LIN {X 0,Y 333.799,Z 297.531,A -85,B 0,C 180,E1 6659.656,E2 6659.656} C_VEL
LIN {X 0,Y 333.556,Z 297.579,A -85,B 0,C 180,E1 6657.079,E2 6657.079} C_VEL
LIN {X 0,Y 335.123,Z 301.286,A -85,B 0,C 180,E1 6651.161,E2 6651.161} C_VEL
LIN {X 0,Y 337.536,Z 305.981,A -85,B 0,C 180,E1 6647.598,E2 6647.598} C_VEL
LIN {X 0,Y 340.159,Z 311.065,A -85,B 0,C 180,E1 6644.834,E2 6644.834} C_VEL
LIN {X 0,Y 343.938,Z 318.214,A -85,B 0,C 180,E1 6641.745,E2 6641.745} C_VEL
LIN {X 0,Y 348.405,Z 327.233,A -85,B 0,C 180,E1 6638.757,E2 6638.757} C_VEL
LIN {X 0,Y 349.368,Z 329.534,A -85,B 0,C 180,E1 6638.161,E2 6638.161} C_VEL
LIN {X 0,Y 333.659,Z 514.335,A -85,B 0,C 180,E1 6634.617,E2 6634.617} C_VEL
LIN {X 0,Y 330.211,Z 536.648,A -85,B 0,C 180,E1 6634.047,E2 6634.047} C_VEL
LIN {X 0,Y 325.459,Z 558.771,A -85,B 0,C 180,E1 6633.278,E2 6633.278} C_VEL
LIN {X 0,Y 319.995,Z 578.663,A -85,B 0,C 180,E1 6632.35,E2 6632.35} C_VEL
LIN {X 0,Y 312.977,Z 599.721,A -85,B 0,C 180,E1 6631.082,E2 6631.082} C_VEL
LIN {X 0,Y 305.406,Z 619.136,A -85,B 0,C 180,E1 6629.614,E2 6629.614} C_VEL
LIN {X 0,Y 297.139,Z 637.32,A -85,B 0,C 180,E1 6627.882,E2 6627.882} C_VEL
LIN {X 0,Y 287.577,Z 656.103,A -85,B 0,C 180,E1 6625.662,E2 6625.662} C_VEL
LIN {X 0,Y 278.286,Z 672.56,A -85,B 0,C 180,E1 6623.245,E2 6623.245} C_VEL
LIN {X 0,Y 268.609,Z 688.083,A -85,B 0,C 180,E1 6620.399,E2 6620.399} C_VEL
LIN {X 0,Y 259.107,Z 702.402,A -85,B 0,C 180,E1 6617.152,E2 6617.152} C_VEL
LIN {X 0,Y 249.96,Z 715.337,A -85,B 0,C 180,E1 6613.471,E2 6613.471} C_VEL
LIN {X 0,Y 241.007,Z 727.524,A -85,B 0,C 180,E1 6609.093,E2 6609.093} C_VEL
LIN {X 0,Y 233.429,Z 737.795,A -85,B 0,C 180,E1 6604.429,E2 6604.429} C_VEL
LIN {X 0,Y 227.015,Z 746.575,A -85,B 0,C 180,E1 6599.266,E2 6599.266} C_VEL
LIN {X 0,Y 222.006,Z 753.904,A -85,B 0,C 180,E1 6593.63,E2 6593.63} C_VEL
LIN {X 0,Y 218.703,Z 759.529,A -85,B 0,C 180,E1 6587.836,E2 6587.836} C_VEL
LIN {X 0,Y 216.939,Z 763.245,A -85,B 0,C 180,E1 6582.24,E2 6582.24} C_VEL
LIN {X 0,Y 216.215,Z 765.602,A -85,B 0,C 180,E1 6576.639,E2 6576.639} C_VEL
LIN {X 0,Y 216.046,Z 766.465,A -85,B 0,C 180,E1 6571.856,E2 6571.856} C_VEL
LIN {X 0,Y 216.061,Z 766.392,A -85,B 0,C 180,E1 6567.082,E2 6567.082} C_VEL
LIN {X 0,Y 216.332,Z 765.111,A -85,B 0,C 180,E1 6561.763,E2 6561.763} C_VEL
LIN {X 0,Y 217.229,Z 762.561,A -85,B 0,C 180,E1 6556.424,E2 6556.424} C_VEL
LIN {X 0,Y 219.54,Z 757.995,A -85,B 0,C 180,E1 6550.305,E2 6550.305} C_VEL
LIN {X 0,Y 223.351,Z 751.966,A -85,B 0,C 180,E1 6544.549,E2 6544.549} C_VEL
LIN {X 0,Y 228.596,Z 744.406,A -85,B 0,C 180,E1 6539.221,E2 6539.221} C_VEL
LIN {X 0,Y 235.447,Z 735.08,A -85,B 0,C 180,E1 6534.125,E2 6534.125} C_VEL
LIN {X 0,Y 243.448,Z 724.408,A -85,B 0,C 180,E1 6529.541,E2 6529.541} C_VEL
LIN {X 0,Y 252.267,Z 712.209,A -85,B 0,C 180,E1 6525.451,E2 6525.451} C_VEL
LIN {X 0,Y 262.23,Z 697.898,A -85,B 0,C 180,E1 6521.642,E2 6521.642} C_VEL
LIN {X 0,Y 272.029,Z 682.985,A -85,B 0,C 180,E1 6518.476,E2 6518.476} C_VEL
LIN {X 0,Y 281.596,Z 667.003,A -85,B 0,C 180,E1 6515.776,E2 6515.776} C_VEL
LIN {X 0,Y 291.404,Z 649.061,A -85,B 0,C 180,E1 6513.335,E2 6513.335} C_VEL
LIN {X 0,Y 300.317,Z 630.949,A -85,B 0,C 180,E1 6511.356,E2 6511.356} C_VEL
LIN {X 0,Y 308.467,Z 611.849,A -85,B 0,C 180,E1 6509.696,E2 6509.696} C_VEL
LIN {X 0,Y 316.13,Z 591.143,A -85,B 0,C 180,E1 6508.259,E2 6508.259} C_VEL
LIN {X 0,Y 322.47,Z 570.714,A -85,B 0,C 180,E1 6507.145,E2 6507.145} C_VEL
LIN {X 0,Y 327.778,Z 549.297,A -85,B 0,C 180,E1 6506.26,E2 6506.26} C_VEL
LIN {X 0,Y 332.035,Z 527,A -85,B 0,C 180,E1 6505.584,E2 6505.584} C_VEL
LIN {X 0,Y 334.766,Z 504.932,A -85,B 0,C 180,E1 6505.085,E2 6505.085} C_VEL
LIN {X 0,Y 335.935,Z 491.115,A -85,B 0,C 180,E1 6504.815,E2 6504.815} C_VEL
LIN {X 0,Y 336.181,Z 483.557,A -85,B 0,C 180,E1 6504.514,E2 6504.514} C_VEL
LIN {X 0,Y 335.511,Z 463.894,A -85,B 0,C 180,E1 6503.143,E2 6503.143} C_VEL
LIN {X 0,Y 335.792,Z 457.395,A -85,B 0,C 180,E1 6502.899,E2 6502.899} C_VEL
LIN {X 0,Y 346.51,Z 334.247,A -85,B 0,C 180,E1 6500.568,E2 6500.568} C_VEL
LIN {X 0,Y 342.284,Z 325.412,A -85,B 0,C 180,E1 6497.598,E2 6497.598} C_VEL
LIN {X 0,Y 338.735,Z 318.442,A -85,B 0,C 180,E1 6494.531,E2 6494.531} C_VEL
LIN {X 0,Y 335.95,Z 312.735,A -85,B 0,C 180,E1 6491.329,E2 6491.329} C_VEL
LIN {X 0,Y 333.881,Z 308.598,A -85,B 0,C 180,E1 6487.745,E2 6487.745} C_VEL
LIN {X 0,Y 332.812,Z 305.703,A -85,B 0,C 180,E1 6482.239,E2 6482.239} C_VEL
LIN {X 0,Y 333.175,Z 306.116,A -85,B 0,C 180,E1 6479.656,E2 6479.656} C_VEL
LIN {X 0,Y 335.748,Z 309.602,A -85,B 0,C 180,E1 6474.275,E2 6474.275} C_VEL
LIN {X 0,Y 338.837,Z 314.734,A -85,B 0,C 180,E1 6470.66,E2 6470.66} C_VEL
LIN {X 0,Y 342.068,Z 320.176,A -85,B 0,C 180,E1 6467.851,E2 6467.851} C_VEL
LIN {X 0,Y 346.16,Z 327.49,A -85,B 0,C 180,E1 6464.933,E2 6464.933} C_VEL
LIN {X 0,Y 348.005,Z 331.065,A -85,B 0,C 180,E1 6463.762,E2 6463.762} C_VEL
LIN {X 0,Y 331.369,Z 511.396,A -85,B 0,C 180,E1 6460.174,E2 6460.174} C_VEL
LIN {X 0,Y 327.681,Z 534.66,A -85,B 0,C 180,E1 6459.571,E2 6459.571} C_VEL
LIN {X 0,Y 322.798,Z 557.073,A -85,B 0,C 180,E1 6458.798,E2 6458.798} C_VEL
LIN {X 0,Y 316.826,Z 578.359,A -85,B 0,C 180,E1 6457.813,E2 6457.813} C_VEL
LIN {X 0,Y 309.169,Z 600.967,A -85,B 0,C 180,E1 6456.465,E2 6456.465} C_VEL
LIN {X 0,Y 301.055,Z 621.475,A -85,B 0,C 180,E1 6454.919,E2 6454.919} C_VEL
LIN {X 0,Y 292.123,Z 640.891,A -85,B 0,C 180,E1 6453.074,E2 6453.074} C_VEL
LIN {X 0,Y 281.948,Z 660.722,A -85,B 0,C 180,E1 6450.733,E2 6450.733} C_VEL
LIN {X 0,Y 272.269,Z 677.831,A -85,B 0,C 180,E1 6448.225,E2 6448.225} C_VEL
LIN {X 0,Y 262.16,Z 694.192,A -85,B 0,C 180,E1 6445.249,E2 6445.249} C_VEL
LIN {X 0,Y 251.99,Z 709.754,A -85,B 0,C 180,E1 6441.759,E2 6441.759} C_VEL
LIN {X 0,Y 242.523,Z 723.441,A -85,B 0,C 180,E1 6437.908,E2 6437.908} C_VEL
LIN {X 0,Y 232.836,Z 737.179,A -85,B 0,C 180,E1 6433.06,E2 6433.06} C_VEL
LIN {X 0,Y 225.094,Z 748.311,A -85,B 0,C 180,E1 6428.128,E2 6428.128} C_VEL
LIN {X 0,Y 218.579,Z 757.937,A -85,B 0,C 180,E1 6422.667,E2 6422.667} C_VEL
LIN {X 0,Y 213.445,Z 766.429,A -85,B 0,C 180,E1 6416.529,E2 6416.529} C_VEL
LIN {X 0,Y 210.416,Z 772.403,A -85,B 0,C 180,E1 6410.878,E2 6410.878} C_VEL
LIN {X 0,Y 208.638,Z 777.202,A -85,B 0,C 180,E1 6404.713,E2 6404.713} C_VEL
LIN {X 0,Y 208.082,Z 779.88,A -85,B 0,C 180,E1 6399.682,E2 6399.682} C_VEL
LIN {X 0,Y 207.995,Z 781.502,A -85,B 0,C 180,E1 6394.687,E2 6394.687} C_VEL
LIN {X 0,Y 208.03,Z 782.018,A -85,B 0,C 180,E1 6389.725,E2 6389.725} C_VEL
LIN {X 0,Y 207.994,Z 781.35,A -85,B 0,C 180,E1 6384.76,E2 6384.76} C_VEL
LIN {X 0,Y 208.096,Z 779.747,A -85,B 0,C 180,E1 6380.04,E2 6380.04} C_VEL
LIN {X 0,Y 208.804,Z 776.674,A -85,B 0,C 180,E1 6374.446,E2 6374.446} C_VEL
LIN {X 0,Y 210.701,Z 771.73,A -85,B 0,C 180,E1 6368.449,E2 6368.449} C_VEL
LIN {X 0,Y 214.139,Z 765.22,A -85,B 0,C 180,E1 6362.468,E2 6362.468} C_VEL
LIN {X 0,Y 219.122,Z 757.046,A -85,B 0,C 180,E1 6356.801,E2 6356.801} C_VEL
LIN {X 0,Y 226.148,Z 746.654,A -85,B 0,C 180,E1 6351.112,E2 6351.112} C_VEL
LIN {X 0,Y 234.128,Z 735.335,A -85,B 0,C 180,E1 6346.226,E2 6346.226} C_VEL
LIN {X 0,Y 243.307,Z 722.206,A -85,B 0,C 180,E1 6341.738,E2 6341.738} C_VEL
LIN {X 0,Y 253.129,Z 707.933,A -85,B 0,C 180,E1 6337.817,E2 6337.817} C_VEL
LIN {X 0,Y 263.1,Z 692.584,A -85,B 0,C 180,E1 6334.448,E2 6334.448} C_VEL
LIN {X 0,Y 273.875,Z 674.84,A -85,B 0,C 180,E1 6331.322,E2 6331.322} C_VEL
LIN {X 0,Y 284.002,Z 656.771,A -85,B 0,C 180,E1 6328.765,E2 6328.765} C_VEL
LIN {X 0,Y 293.417,Z 637.944,A -85,B 0,C 180,E1 6326.636,E2 6326.636} C_VEL
LIN {X 0,Y 302.733,Z 617.038,A -85,B 0,C 180,E1 6324.737,E2 6324.737} C_VEL
LIN {X 0,Y 310.741,Z 596.454,A -85,B 0,C 180,E1 6323.244,E2 6323.244} C_VEL
LIN {X 0,Y 317.653,Z 575.154,A -85,B 0,C 180,E1 6322.035,E2 6322.035} C_VEL
LIN {X 0,Y 323.863,Z 551.917,A -85,B 0,C 180,E1 6321.013,E2 6321.013} C_VEL
LIN {X 0,Y 328.488,Z 529.683,A -85,B 0,C 180,E1 6320.29,E2 6320.29} C_VEL
LIN {X 0,Y 331.75,Z 506.604,A -85,B 0,C 180,E1 6319.732,E2 6319.732} C_VEL
LIN {X 0,Y 347.863,Z 330.818,A -85,B 0,C 180,E1 6316.238,E2 6316.238} C_VEL
LIN {X 0,Y 343.256,Z 322.384,A -85,B 0,C 180,E1 6313.175,E2 6313.175} C_VEL
LIN {X 0,Y 339.741,Z 316.374,A -85,B 0,C 180,E1 6310.342,E2 6310.342} C_VEL
LIN {X 0,Y 337.54,Z 312.774,A -85,B 0,C 180,E1 6308.174,E2 6308.174} C_VEL
LIN {X 0,Y 335.255,Z 309.045,A -85,B 0,C 180,E1 6305.305,E2 6305.305} C_VEL
LIN {X 0,Y 332.793,Z 305.429,A -85,B 0,C 180,E1 6299.483,E2 6299.483} C_VEL
LIN {X 0,Y 332.58,Z 305.538,A -85,B 0,C 180,E1 6297.07,E2 6297.07} C_VEL
LIN {X 0,Y 334.018,Z 309.105,A -85,B 0,C 180,E1 6291.392,E2 6291.392} C_VEL
LIN {X 0,Y 336.286,Z 313.689,A -85,B 0,C 180,E1 6287.9,E2 6287.9} C_VEL
LIN {X 0,Y 338.827,Z 318.787,A -85,B 0,C 180,E1 6285.124,E2 6285.124} C_VEL
LIN {X 0,Y 342.557,Z 326.138,A -85,B 0,C 180,E1 6281.977,E2 6281.977} C_VEL
LIN {X 0,Y 346.368,Z 334.145,A -85,B 0,C 180,E1 6279.331,E2 6279.331} C_VEL
LIN {X 0,Y 330.595,Z 514.238,A -85,B 0,C 180,E1 6275.897,E2 6275.897} C_VEL
LIN {X 0,Y 327.044,Z 536.692,A -85,B 0,C 180,E1 6275.332,E2 6275.332} C_VEL
LIN {X 0,Y 322.156,Z 558.903,A -85,B 0,C 180,E1 6274.573,E2 6274.573} C_VEL
LIN {X 0,Y 316.376,Z 579.413,A -85,B 0,C 180,E1 6273.629,E2 6273.629} C_VEL
LIN {X 0,Y 309.189,Z 600.314,A -85,B 0,C 180,E1 6272.38,E2 6272.38} C_VEL
LIN {X 0,Y 301.428,Z 619.632,A -85,B 0,C 180,E1 6270.93,E2 6270.93} C_VEL
LIN {X 0,Y 292.82,Z 638.021,A -85,B 0,C 180,E1 6269.19,E2 6269.19} C_VEL
LIN {X 0,Y 282.759,Z 657.106,A -85,B 0,C 180,E1 6266.932,E2 6266.932} C_VEL
LIN {X 0,Y 272.873,Z 674.008,A -85,B 0,C 180,E1 6264.432,E2 6264.432} C_VEL
LIN {X 0,Y 262.899,Z 689.345,A -85,B 0,C 180,E1 6261.576,E2 6261.576} C_VEL
LIN {X 0,Y 252.519,Z 704.237,A -85,B 0,C 180,E1 6258.105,E2 6258.105} C_VEL
LIN {X 0,Y 242.805,Z 717.433,A -85,B 0,C 180,E1 6254.231,E2 6254.231} C_VEL
LIN {X 0,Y 233.844,Z 728.953,A -85,B 0,C 180,E1 6249.892,E2 6249.892} C_VEL
LIN {X 0,Y 225.636,Z 739.428,A -85,B 0,C 180,E1 6244.863,E2 6244.863} C_VEL
LIN {X 0,Y 219.071,Z 748.046,A -85,B 0,C 180,E1 6239.532,E2 6239.532} C_VEL
LIN {X 0,Y 213.953,Z 755.074,A -85,B 0,C 180,E1 6233.696,E2 6233.696} C_VEL
LIN {X 0,Y 210.496,Z 760.607,A -85,B 0,C 180,E1 6227.412,E2 6227.412} C_VEL
LIN {X 0,Y 208.819,Z 764.143,A -85,B 0,C 180,E1 6221.601,E2 6221.601} C_VEL
LIN {X 0,Y 208.183,Z 766.083,A -85,B 0,C 180,E1 6216.065,E2 6216.065} C_VEL
LIN {X 0,Y 208.05,Z 766.82,A -85,B 0,C 180,E1 6211.101,E2 6211.101} C_VEL
LIN {X 0,Y 208.1,Z 766.558,A -85,B 0,C 180,E1 6205.867,E2 6205.867} C_VEL
LIN {X 0,Y 208.5,Z 764.977,A -85,B 0,C 180,E1 6200.338,E2 6200.338} C_VEL
LIN {X 0,Y 209.774,Z 762.063,A -85,B 0,C 180,E1 6194.52,E2 6194.52} C_VEL
LIN {X 0,Y 212.497,Z 757.324,A -85,B 0,C 180,E1 6188.469,E2 6188.469} C_VEL
LIN {X 0,Y 216.927,Z 750.912,A -85,B 0,C 180,E1 6182.554,E2 6182.554} C_VEL
LIN {X 0,Y 223.082,Z 742.845,A -85,B 0,C 180,E1 6176.945,E2 6176.945} C_VEL
LIN {X 0,Y 230.422,Z 733.396,A -85,B 0,C 180,E1 6171.964,E2 6171.964} C_VEL
LIN {X 0,Y 239.579,Z 721.646,A -85,B 0,C 180,E1 6167.137,E2 6167.137} C_VEL
LIN {X 0,Y 249.147,Z 709.054,A -85,B 0,C 180,E1 6163.083,E2 6163.083} C_VEL
LIN {X 0,Y 258.622,Z 695.757,A -85,B 0,C 180,E1 6159.706,E2 6159.706} C_VEL
LIN {X 0,Y 269.416,Z 679.56,A -85,B 0,C 180,E1 6156.427,E2 6156.427} C_VEL
LIN {X 0,Y 279.594,Z 662.962,A -85,B 0,C 180,E1 6153.755,E2 6153.755} C_VEL
LIN {X 0,Y 289.138,Z 645.535,A -85,B 0,C 180,E1 6151.527,E2 6151.527} C_VEL
LIN {X 0,Y 298.371,Z 626.661,A -85,B 0,C 180,E1 6149.591,E2 6149.591} C_VEL
LIN {X 0,Y 306.714,Z 607.269,A -85,B 0,C 180,E1 6147.997,E2 6147.997} C_VEL
LIN {X 0,Y 313.949,Z 587.306,A -85,B 0,C 180,E1 6146.708,E2 6146.708} C_VEL
LIN {X 0,Y 320.465,Z 565.899,A -85,B 0,C 180,E1 6145.623,E2 6145.623} C_VEL
LIN {X 0,Y 325.353,Z 545.873,A -85,B 0,C 180,E1 6144.851,E2 6144.851} C_VEL
LIN {X 0,Y 329.463,Z 523.359,A -85,B 0,C 180,E1 6144.215,E2 6144.215} C_VEL
LIN {X 0,Y 332.202,Z 499.849,A -85,B 0,C 180,E1 6143.708,E2 6143.708} C_VEL
LIN {X 0,Y 335.792,Z 457.395,A -85,B 0,C 180,E1 6142.899,E2 6142.899} C_VEL
LIN {X 0,Y 336.087,Z 449.841,A -85,B 0,C 180,E1 6142.594,E2 6142.594} C_VEL
LIN {X 0,Y 335.695,Z 430.195,A -85,B 0,C 180,E1 6141.211,E2 6141.211} C_VEL
LIN {X 0,Y 336.035,Z 423.697,A -85,B 0,C 180,E1 6140.971,E2 6140.971} C_VEL
LIN {X 0,Y 343.619,Z 339.193,A -85,B 0,C 180,E1 6139.373,E2 6139.373} C_VEL
LIN {X 0,Y 339.767,Z 330.925,A -85,B 0,C 180,E1 6136.41,E2 6136.41} C_VEL
LIN {X 0,Y 336.405,Z 323.949,A -85,B 0,C 180,E1 6133.143,E2 6133.143} C_VEL
LIN {X 0,Y 334.367,Z 319.872,A -85,B 0,C 180,E1 6130.51,E2 6130.51} C_VEL
LIN {X 0,Y 332.808,Z 316.439,A -85,B 0,C 180,E1 6127.522,E2 6127.522} C_VEL
LIN {X 0,Y 331.836,Z 313.655,A -85,B 0,C 180,E1 6122.245,E2 6122.245} C_VEL
LIN {X 0,Y 332.158,Z 313.997,A -85,B 0,C 180,E1 6119.828,E2 6119.828} C_VEL
LIN {X 0,Y 334.577,Z 317.402,A -85,B 0,C 180,E1 6114.513,E2 6114.513} C_VEL
LIN {X 0,Y 337.577,Z 322.568,A -85,B 0,C 180,E1 6110.883,E2 6110.883} C_VEL
LIN {X 0,Y 340.629,Z 327.878,A -85,B 0,C 180,E1 6108.143,E2 6108.143} C_VEL
LIN {X 0,Y 344.745,Z 335.474,A -85,B 0,C 180,E1 6105.127,E2 6105.127} C_VEL
LIN {X 0,Y 345.018,Z 336.358,A -85,B 0,C 180,E1 6104.922,E2 6104.922} C_VEL
LIN {X 0,Y 328.43,Z 511.584,A -85,B 0,C 180,E1 6101.468,E2 6101.468} C_VEL
LIN {X 0,Y 324.675,Z 534.746,A -85,B 0,C 180,E1 6100.878,E2 6100.878} C_VEL
LIN {X 0,Y 319.704,Z 557.076,A -85,B 0,C 180,E1 6100.124,E2 6100.124} C_VEL
LIN {X 0,Y 313.499,Z 578.698,A -85,B 0,C 180,E1 6099.14,E2 6099.14} C_VEL
LIN {X 0,Y 305.987,Z 600.374,A -85,B 0,C 180,E1 6097.873,E2 6097.873} C_VEL
LIN {X 0,Y 297.498,Z 621.33,A -85,B 0,C 180,E1 6096.322,E2 6096.322} C_VEL
LIN {X 0,Y 288.555,Z 640.271,A -85,B 0,C 180,E1 6094.554,E2 6094.554} C_VEL
LIN {X 0,Y 278.341,Z 659.691,A -85,B 0,C 180,E1 6092.307,E2 6092.307} C_VEL
LIN {X 0,Y 268.308,Z 676.872,A -85,B 0,C 180,E1 6089.829,E2 6089.829} C_VEL
LIN {X 0,Y 257.656,Z 693.579,A -85,B 0,C 180,E1 6086.828,E2 6086.828} C_VEL
LIN {X 0,Y 247.511,Z 708.558,A -85,B 0,C 180,E1 6083.501,E2 6083.501} C_VEL
LIN {X 0,Y 236.977,Z 723.105,A -85,B 0,C 180,E1 6079.415,E2 6079.415} C_VEL
LIN {X 0,Y 226.773,Z 736.859,A -85,B 0,C 180,E1 6074.509,E2 6074.509} C_VEL
LIN {X 0,Y 218.548,Z 747.992,A -85,B 0,C 180,E1 6069.487,E2 6069.487} C_VEL
LIN {X 0,Y 211.578,Z 757.626,A -85,B 0,C 180,E1 6063.891,E2 6063.891} C_VEL
LIN {X 0,Y 206.155,Z 765.916,A -85,B 0,C 180,E1 6057.748,E2 6057.748} C_VEL
LIN {X 0,Y 202.844,Z 771.832,A -85,B 0,C 180,E1 6052,E2 6052} C_VEL
LIN {X 0,Y 200.741,Z 776.906,A -85,B 0,C 180,E1 6045.306,E2 6045.306} C_VEL
LIN {X 0,Y 200.102,Z 779.586,A -85,B 0,C 180,E1 6040.072,E2 6040.072} C_VEL
LIN {X 0,Y 199.997,Z 781.211,A -85,B 0,C 180,E1 6034.875,E2 6034.875} C_VEL
LIN {X 0,Y 200.035,Z 781.727,A -85,B 0,C 180,E1 6029.714,E2 6029.714} C_VEL
LIN {X 0,Y 199.997,Z 781.058,A -85,B 0,C 180,E1 6024.55,E2 6024.55} C_VEL
LIN {X 0,Y 200.12,Z 779.451,A -85,B 0,C 180,E1 6019.638,E2 6019.638} C_VEL
LIN {X 0,Y 200.923,Z 776.376,A -85,B 0,C 180,E1 6013.819,E2 6013.819} C_VEL
LIN {X 0,Y 202.97,Z 771.536,A -85,B 0,C 180,E1 6007.71,E2 6007.71} C_VEL
LIN {X 0,Y 206.57,Z 765.244,A -85,B 0,C 180,E1 6001.684,E2 6001.684} C_VEL
LIN {X 0,Y 211.866,Z 757.155,A -85,B 0,C 180,E1 5995.835,E2 5995.835} C_VEL
LIN {X 0,Y 218.913,Z 747.401,A -85,B 0,C 180,E1 5990.252,E2 5990.252} C_VEL
LIN {X 0,Y 227.219,Z 736.196,A -85,B 0,C 180,E1 5985.247,E2 5985.247} C_VEL
LIN {X 0,Y 237.229,Z 722.653,A -85,B 0,C 180,E1 5980.471,E2 5980.471} C_VEL
LIN {X 0,Y 247.5,Z 708.444,A -85,B 0,C 180,E1 5976.495,E2 5976.495} C_VEL
LIN {X 0,Y 257.831,Z 693.165,A -85,B 0,C 180,E1 5973.111,E2 5973.111} C_VEL
LIN {X 0,Y 269.302,Z 675.009,A -85,B 0,C 180,E1 5969.899,E2 5969.899} C_VEL
LIN {X 0,Y 279.396,Z 657.645,A -85,B 0,C 180,E1 5967.442,E2 5967.442} C_VEL
LIN {X 0,Y 289.323,Z 638.454,A -85,B 0,C 180,E1 5965.277,E2 5965.277} C_VEL
LIN {X 0,Y 298.891,Z 617.672,A -85,B 0,C 180,E1 5963.402,E2 5963.402} C_VEL
LIN {X 0,Y 307.154,Z 597.004,A -85,B 0,C 180,E1 5961.918,E2 5961.918} C_VEL
LIN {X 0,Y 314.28,Z 575.687,A -85,B 0,C 180,E1 5960.721,E2 5960.721} C_VEL
LIN {X 0,Y 320.498,Z 553.187,A -85,B 0,C 180,E1 5959.738,E2 5959.738} C_VEL
LIN {X 0,Y 325.186,Z 531.346,A -85,B 0,C 180,E1 5959.032,E2 5959.032} C_VEL
LIN {X 0,Y 328.718,Z 507.683,A -85,B 0,C 180,E1 5958.459,E2 5958.459} C_VEL
LIN {X 0,Y 344.865,Z 335.93,A -85,B 0,C 180,E1 5955.064,E2 5955.064} C_VEL
LIN {X 0,Y 340.775,Z 328.253,A -85,B 0,C 180,E1 5952.11,E2 5952.11} C_VEL
LIN {X 0,Y 337.662,Z 322.863,A -85,B 0,C 180,E1 5949.373,E2 5949.373} C_VEL
LIN {X 0,Y 335.93,Z 320.014,A -85,B 0,C 180,E1 5947.525,E2 5947.525} C_VEL
LIN {X 0,Y 334.034,Z 316.781,A -85,B 0,C 180,E1 5944.98,E2 5944.98} C_VEL
LIN {X 0,Y 331.789,Z 313.328,A -85,B 0,C 180,E1 5939.309,E2 5939.309} C_VEL
LIN {X 0,Y 331.602,Z 313.552,A -85,B 0,C 180,E1 5936.955,E2 5936.955} C_VEL
LIN {X 0,Y 332.92,Z 316.923,A -85,B 0,C 180,E1 5931.624,E2 5931.624} C_VEL
LIN {X 0,Y 335.067,Z 321.465,A -85,B 0,C 180,E1 5928.165,E2 5928.165} C_VEL
LIN {X 0,Y 337.851,Z 327.149,A -85,B 0,C 180,E1 5925.08,E2 5925.08} C_VEL
LIN {X 0,Y 341.177,Z 334.101,A -85,B 0,C 180,E1 5922.21,E2 5922.21} C_VEL
LIN {X 0,Y 343.483,Z 339.338,A -85,B 0,C 180,E1 5920.5,E2 5920.5} C_VEL
LIN {X 0,Y 327.692,Z 514.168,A -85,B 0,C 180,E1 5917.199,E2 5917.199} C_VEL
LIN {X 0,Y 324.064,Z 536.634,A -85,B 0,C 180,E1 5916.645,E2 5916.645} C_VEL
LIN {X 0,Y 319.02,Z 559.031,A -85,B 0,C 180,E1 5915.895,E2 5915.895} C_VEL
LIN {X 0,Y 313.304,Z 578.886,A -85,B 0,C 180,E1 5915.001,E2 5915.001} C_VEL
LIN {X 0,Y 305.946,Z 599.91,A -85,B 0,C 180,E1 5913.775,E2 5913.775} C_VEL
LIN {X 0,Y 297.989,Z 619.319,A -85,B 0,C 180,E1 5912.349,E2 5912.349} C_VEL
LIN {X 0,Y 289.115,Z 637.808,A -85,B 0,C 180,E1 5910.631,E2 5910.631} C_VEL
LIN {X 0,Y 278.971,Z 656.588,A -85,B 0,C 180,E1 5908.447,E2 5908.447} C_VEL
LIN {X 0,Y 268.903,Z 673.331,A -85,B 0,C 180,E1 5906.012,E2 5906.012} C_VEL
LIN {X 0,Y 258.528,Z 688.828,A -85,B 0,C 180,E1 5903.168,E2 5903.168} C_VEL
LIN {X 0,Y 247.721,Z 703.818,A -85,B 0,C 180,E1 5899.714,E2 5899.714} C_VEL
LIN {X 0,Y 237.84,Z 716.674,A -85,B 0,C 180,E1 5895.96,E2 5895.96} C_VEL
LIN {X 0,Y 228.528,Z 728.154,A -85,B 0,C 180,E1 5891.683,E2 5891.683} C_VEL
LIN {X 0,Y 220.104,Z 738.408,A -85,B 0,C 180,E1 5886.842,E2 5886.842} C_VEL
LIN {X 0,Y 212.871,Z 747.186,A -85,B 0,C 180,E1 5881.423,E2 5881.423} C_VEL
LIN {X 0,Y 207.136,Z 754.504,A -85,B 0,C 180,E1 5875.442,E2 5875.442} C_VEL
LIN {X 0,Y 203.268,Z 760.122,A -85,B 0,C 180,E1 5869.242,E2 5869.242} C_VEL
LIN {X 0,Y 201.156,Z 763.836,A -85,B 0,C 180,E1 5863.217,E2 5863.217} C_VEL
LIN {X 0,Y 200.244,Z 766.248,A -85,B 0,C 180,E1 5856.882,E2 5856.882} C_VEL
LIN {X 0,Y 200.057,Z 767.072,A -85,B 0,C 180,E1 5851.66,E2 5851.66} C_VEL
LIN {X 0,Y 200.084,Z 766.953,A -85,B 0,C 180,E1 5846.562,E2 5846.562} C_VEL
LIN {X 0,Y 200.446,Z 765.589,A -85,B 0,C 180,E1 5840.815,E2 5840.815} C_VEL
LIN {X 0,Y 201.594,Z 762.998,A -85,B 0,C 180,E1 5835.054,E2 5835.054} C_VEL
LIN {X 0,Y 204.259,Z 758.589,A -85,B 0,C 180,E1 5828.763,E2 5828.763} C_VEL
LIN {X 0,Y 208.692,Z 752.568,A -85,B 0,C 180,E1 5822.617,E2 5822.617} C_VEL
LIN {X 0,Y 214.701,Z 744.975,A -85,B 0,C 180,E1 5816.957,E2 5816.957} C_VEL
LIN {X 0,Y 222.774,Z 735.198,A -85,B 0,C 180,E1 5811.403,E2 5811.403} C_VEL
LIN {X 0,Y 231.704,Z 724.431,A -85,B 0,C 180,E1 5806.678,E2 5806.678} C_VEL
LIN {X 0,Y 241.435,Z 712.168,A -85,B 0,C 180,E1 5802.512,E2 5802.512} C_VEL
LIN {X 0,Y 251.697,Z 698.574,A -85,B 0,C 180,E1 5798.869,E2 5798.869} C_VEL
LIN {X 0,Y 262.271,Z 683.632,A -85,B 0,C 180,E1 5795.682,E2 5795.682} C_VEL
LIN {X 0,Y 272.782,Z 667.21,A -85,B 0,C 180,E1 5792.928,E2 5792.928} C_VEL
LIN {X 0,Y 283.216,Z 649.242,A -85,B 0,C 180,E1 5790.527,E2 5790.527} C_VEL
LIN {X 0,Y 292.828,Z 630.745,A -85,B 0,C 180,E1 5788.557,E2 5788.557} C_VEL
LIN {X 0,Y 301.231,Z 612.009,A -85,B 0,C 180,E1 5786.977,E2 5786.977} C_VEL
LIN {X 0,Y 309.278,Z 591.313,A -85,B 0,C 180,E1 5785.585,E2 5785.585} C_VEL
LIN {X 0,Y 315.519,Z 572.179,A -85,B 0,C 180,E1 5784.569,E2 5784.569} C_VEL
LIN {X 0,Y 321.306,Z 550.248,A -85,B 0,C 180,E1 5783.68,E2 5783.68} C_VEL
LIN {X 0,Y 325.784,Z 528.283,A -85,B 0,C 180,E1 5783.028,E2 5783.028} C_VEL
LIN {X 0,Y 328.747,Z 505.867,A -85,B 0,C 180,E1 5782.529,E2 5782.529} C_VEL
LIN {X 0,Y 336.035,Z 423.697,A -85,B 0,C 180,E1 5780.971,E2 5780.971} C_VEL
LIN {X 0,Y 336.398,Z 416.144,A -85,B 0,C 180,E1 5780.671,E2 5780.671} C_VEL
LIN {X 0,Y 336.265,Z 396.516,A -85,B 0,C 180,E1 5779.282,E2 5779.282} C_VEL
LIN {X 0,Y 336.643,Z 390.022,A -85,B 0,C 180,E1 5779.038,E2 5779.038} C_VEL
LIN {X 0,Y 340.866,Z 344.206,A -85,B 0,C 180,E1 5778.16,E2 5778.16} C_VEL
LIN {X 0,Y 337.728,Z 337.382,A -85,B 0,C 180,E1 5775.541,E2 5775.541} C_VEL
LIN {X 0,Y 334.984,Z 331.384,A -85,B 0,C 180,E1 5772.673,E2 5772.673} C_VEL
LIN {X 0,Y 333.17,Z 327.584,A -85,B 0,C 180,E1 5770.199,E2 5770.199} C_VEL
LIN {X 0,Y 331.723,Z 324.266,A -85,B 0,C 180,E1 5767.273,E2 5767.273} C_VEL
LIN {X 0,Y 330.873,Z 321.562,A -85,B 0,C 180,E1 5762.078,E2 5762.078} C_VEL
LIN {X 0,Y 331.25,Z 322.126,A -85,B 0,C 180,E1 5759.481,E2 5759.481} C_VEL
LIN {X 0,Y 333.465,Z 325.323,A -85,B 0,C 180,E1 5754.667,E2 5754.667} C_VEL
LIN {X 0,Y 336.242,Z 330.251,A -85,B 0,C 180,E1 5751.191,E2 5751.191} C_VEL
LIN {X 0,Y 339.197,Z 335.579,A -85,B 0,C 180,E1 5748.437,E2 5748.437} C_VEL
LIN {X 0,Y 342.193,Z 341.477,A -85,B 0,C 180,E1 5746.105,E2 5746.105} C_VEL
LIN {X 0,Y 325.674,Z 511.674,A -85,B 0,C 180,E1 5742.787,E2 5742.787} C_VEL
LIN {X 0,Y 321.84,Z 534.834,A -85,B 0,C 180,E1 5742.208,E2 5742.208} C_VEL
LIN {X 0,Y 316.721,Z 557.318,A -85,B 0,C 180,E1 5741.464,E2 5741.464} C_VEL
LIN {X 0,Y 310.684,Z 577.955,A -85,B 0,C 180,E1 5740.548,E2 5740.548} C_VEL
LIN {X 0,Y 302.596,Z 600.8,A -85,B 0,C 180,E1 5739.241,E2 5739.241} C_VEL
LIN {X 0,Y 294.291,Z 620.797,A -85,B 0,C 180,E1 5737.789,E2 5737.789} C_VEL
LIN {X 0,Y 285.025,Z 639.97,A -85,B 0,C 180,E1 5736.036,E2 5736.036} C_VEL
LIN {X 0,Y 274.753,Z 659.006,A -85,B 0,C 180,E1 5733.875,E2 5733.875} C_VEL
LIN {X 0,Y 264.222,Z 676.482,A -85,B 0,C 180,E1 5731.39,E2 5731.39} C_VEL
LIN {X 0,Y 253.047,Z 693.41,A -85,B 0,C 180,E1 5728.373,E2 5728.373} C_VEL
LIN {X 0,Y 242.016,Z 709.037,A -85,B 0,C 180,E1 5724.884,E2 5724.884} C_VEL
LIN {X 0,Y 231.31,Z 723.162,A -85,B 0,C 180,E1 5720.869,E2 5720.869} C_VEL
LIN {X 0,Y 220.86,Z 736.537,A -85,B 0,C 180,E1 5716.037,E2 5716.037} C_VEL
LIN {X 0,Y 212.13,Z 747.673,A -85,B 0,C 180,E1 5710.931,E2 5710.931} C_VEL
LIN {X 0,Y 204.677,Z 757.314,A -85,B 0,C 180,E1 5705.199,E2 5705.199} C_VEL
LIN {X 0,Y 198.818,Z 765.612,A -85,B 0,C 180,E1 5698.867,E2 5698.867} C_VEL
LIN {X 0,Y 195.1,Z 771.707,A -85,B 0,C 180,E1 5692.711,E2 5692.711} C_VEL
LIN {X 0,Y 192.859,Z 776.608,A -85,B 0,C 180,E1 5685.948,E2 5685.948} C_VEL
LIN {X 0,Y 192.122,Z 779.333,A -85,B 0,C 180,E1 5680.391,E2 5680.391} C_VEL
LIN {X 0,Y 192.001,Z 780.919,A -85,B 0,C 180,E1 5675.079,E2 5675.079} C_VEL
LIN {X 0,Y 192.04,Z 781.437,A -85,B 0,C 180,E1 5669.702,E2 5669.702} C_VEL
LIN {X 0,Y 192.003,Z 780.765,A -85,B 0,C 180,E1 5664.322,E2 5664.322} C_VEL
LIN {X 0,Y 192.15,Z 779.156,A -85,B 0,C 180,E1 5659.203,E2 5659.203} C_VEL
LIN {X 0,Y 193.061,Z 776.077,A -85,B 0,C 180,E1 5653.141,E2 5653.141} C_VEL
LIN {X 0,Y 195.335,Z 771.232,A -85,B 0,C 180,E1 5646.788,E2 5646.788} C_VEL
LIN {X 0,Y 199.502,Z 764.6,A -85,B 0,C 180,E1 5640.254,E2 5640.254} C_VEL
LIN {X 0,Y 205.304,Z 756.419,A -85,B 0,C 180,E1 5634.239,E2 5634.239} C_VEL
LIN {X 0,Y 213.329,Z 746.011,A -85,B 0,C 180,E1 5628.277,E2 5628.277} C_VEL
LIN {X 0,Y 222.29,Z 734.686,A -85,B 0,C 180,E1 5623.226,E2 5623.226} C_VEL
LIN {X 0,Y 232.148,Z 721.954,A -85,B 0,C 180,E1 5618.781,E2 5618.781} C_VEL
LIN {X 0,Y 242.611,Z 708.087,A -85,B 0,C 180,E1 5614.905,E2 5614.905} C_VEL
LIN {X 0,Y 253.361,Z 692.8,A -85,B 0,C 180,E1 5611.527,E2 5611.527} C_VEL
LIN {X 0,Y 265.149,Z 674.785,A -85,B 0,C 180,E1 5608.368,E2 5608.368} C_VEL
LIN {X 0,Y 275.678,Z 657.227,A -85,B 0,C 180,E1 5605.914,E2 5605.914} C_VEL
LIN {X 0,Y 285.772,Z 638.233,A -85,B 0,C 180,E1 5603.807,E2 5603.807} C_VEL
LIN {X 0,Y 295.842,Z 616.85,A -85,B 0,C 180,E1 5601.921,E2 5601.921} C_VEL
LIN {X 0,Y 304.195,Z 596.402,A -85,B 0,C 180,E1 5600.489,E2 5600.489} C_VEL
LIN {X 0,Y 311.486,Z 574.931,A -85,B 0,C 180,E1 5599.317,E2 5599.317} C_VEL
LIN {X 0,Y 317.988,Z 551.533,A -85,B 0,C 180,E1 5598.333,E2 5598.333} C_VEL
LIN {X 0,Y 322.851,Z 528.982,A -85,B 0,C 180,E1 5597.636,E2 5597.636} C_VEL
LIN {X 0,Y 326.173,Z 505.964,A -85,B 0,C 180,E1 5597.103,E2 5597.103} C_VEL
LIN {X 0,Y 342.026,Z 341.243,A -85,B 0,C 180,E1 5593.89,E2 5593.89} C_VEL
LIN {X 0,Y 338.444,Z 334.385,A -85,B 0,C 180,E1 5591.071,E2 5591.071} C_VEL
LIN {X 0,Y 335.302,Z 328.678,A -85,B 0,C 180,E1 5587.97,E2 5587.97} C_VEL
LIN {X 0,Y 332.934,Z 324.653,A -85,B 0,C 180,E1 5584.823,E2 5584.823} C_VEL
LIN {X 0,Y 330.813,Z 321.277,A -85,B 0,C 180,E1 5579.307,E2 5579.307} C_VEL
LIN {X 0,Y 330.626,Z 321.472,A -85,B 0,C 180,E1 5577.053,E2 5577.053} C_VEL
LIN {X 0,Y 331.862,Z 324.857,A -85,B 0,C 180,E1 5571.772,E2 5571.772} C_VEL
LIN {X 0,Y 333.8,Z 329.103,A -85,B 0,C 180,E1 5568.51,E2 5568.51} C_VEL
LIN {X 0,Y 336.521,Z 334.865,A -85,B 0,C 180,E1 5565.371,E2 5565.371} C_VEL
LIN {X 0,Y 339.644,Z 341.745,A -85,B 0,C 180,E1 5562.57,E2 5562.57} C_VEL
LIN {X 0,Y 340.732,Z 344.478,A -85,B 0,C 180,E1 5561.696,E2 5561.696} C_VEL
LIN {X 0,Y 324.968,Z 514.053,A -85,B 0,C 180,E1 5558.525,E2 5558.525} C_VEL
LIN {X 0,Y 321.257,Z 536.567,A -85,B 0,C 180,E1 5557.981,E2 5557.981} C_VEL
LIN {X 0,Y 316.26,Z 558.423,A -85,B 0,C 180,E1 5557.271,E2 5557.271} C_VEL
LIN {X 0,Y 310.416,Z 578.356,A -85,B 0,C 180,E1 5556.399,E2 5556.399} C_VEL
LIN {X 0,Y 302.89,Z 599.504,A -85,B 0,C 180,E1 5555.198,E2 5555.198} C_VEL
LIN {X 0,Y 294.776,Z 618.901,A -85,B 0,C 180,E1 5553.807,E2 5553.807} C_VEL
LIN {X 0,Y 285.785,Z 637.229,A -85,B 0,C 180,E1 5552.144,E2 5552.144} C_VEL
LIN {X 0,Y 275.357,Z 656.115,A -85,B 0,C 180,E1 5549.997,E2 5549.997} C_VEL
LIN {X 0,Y 265.142,Z 672.624,A -85,B 0,C 180,E1 5547.638,E2 5547.638} C_VEL
LIN {X 0,Y 254.416,Z 688.236,A -85,B 0,C 180,E1 5544.827,E2 5544.827} C_VEL
LIN {X 0,Y 243.74,Z 702.644,A -85,B 0,C 180,E1 5541.581,E2 5541.581} C_VEL
LIN {X 0,Y 233.321,Z 715.635,A -85,B 0,C 180,E1 5537.846,E2 5537.846} C_VEL
LIN {X 0,Y 222.962,Z 727.912,A -85,B 0,C 180,E1 5533.322,E2 5533.322} C_VEL
LIN {X 0,Y 214.01,Z 738.27,A -85,B 0,C 180,E1 5528.416,E2 5528.416} C_VEL
LIN {X 0,Y 206.246,Z 747.101,A -85,B 0,C 180,E1 5522.885,E2 5522.885} C_VEL
LIN {X 0,Y 200.019,Z 754.515,A -85,B 0,C 180,E1 5516.736,E2 5516.736} C_VEL
LIN {X 0,Y 195.749,Z 760.222,A -85,B 0,C 180,E1 5510.324,E2 5510.324} C_VEL
LIN {X 0,Y 193.358,Z 763.979,A -85,B 0,C 180,E1 5504.065,E2 5504.065} C_VEL
LIN {X 0,Y 192.322,Z 766.415,A -85,B 0,C 180,E1 5497.768,E2 5497.768} C_VEL
LIN {X 0,Y 192.066,Z 767.338,A -85,B 0,C 180,E1 5492.088,E2 5492.088} C_VEL
LIN {X 0,Y 192.078,Z 767.285,A -85,B 0,C 180,E1 5487.016,E2 5487.016} C_VEL
LIN {X 0,Y 192.425,Z 766.096,A -85,B 0,C 180,E1 5481.032,E2 5481.032} C_VEL
LIN {X 0,Y 193.609,Z 763.555,A -85,B 0,C 180,E1 5474.958,E2 5474.958} C_VEL
LIN {X 0,Y 196.506,Z 759.129,A -85,B 0,C 180,E1 5468.196,E2 5468.196} C_VEL
LIN {X 0,Y 201.198,Z 753.188,A -85,B 0,C 180,E1 5461.83,E2 5461.83} C_VEL
LIN {X 0,Y 207.61,Z 745.578,A -85,B 0,C 180,E1 5455.931,E2 5455.931} C_VEL
LIN {X 0,Y 216.323,Z 735.627,A -85,B 0,C 180,E1 5450.109,E2 5450.109} C_VEL
LIN {X 0,Y 225.816,Z 724.748,A -85,B 0,C 180,E1 5445.252,E2 5445.252} C_VEL
LIN {X 0,Y 236,Z 712.479,A -85,B 0,C 180,E1 5441.048,E2 5441.048} C_VEL
LIN {X 0,Y 247.283,Z 698.084,A -85,B 0,C 180,E1 5437.201,E2 5437.201} C_VEL
LIN {X 0,Y 258.232,Z 683.079,A -85,B 0,C 180,E1 5434.048,E2 5434.048} C_VEL
LIN {X 0,Y 268.965,Z 666.813,A -85,B 0,C 180,E1 5431.362,E2 5431.362} C_VEL
LIN {X 0,Y 279.574,Z 649.001,A -85,B 0,C 180,E1 5429.026,E2 5429.026} C_VEL
LIN {X 0,Y 289.264,Z 630.82,A -85,B 0,C 180,E1 5427.122,E2 5427.122} C_VEL
LIN {X 0,Y 298.072,Z 611.64,A -85,B 0,C 180,E1 5425.536,E2 5425.536} C_VEL
LIN {X 0,Y 306.311,Z 590.834,A -85,B 0,C 180,E1 5424.173,E2 5424.173} C_VEL
LIN {X 0,Y 313.032,Z 570.585,A -85,B 0,C 180,E1 5423.134,E2 5423.134} C_VEL
LIN {X 0,Y 318.632,Z 549.413,A -85,B 0,C 180,E1 5422.31,E2 5422.31} C_VEL
LIN {X 0,Y 323.172,Z 527.21,A -85,B 0,C 180,E1 5421.674,E2 5421.674} C_VEL
LIN {X 0,Y 326.128,Z 505.091,A -85,B 0,C 180,E1 5421.192,E2 5421.192} C_VEL
LIN {X 0,Y 336.643,Z 390.022,A -85,B 0,C 180,E1 5419.038,E2 5419.038} C_VEL
LIN {X 0,Y 337.059,Z 382.472,A -85,B 0,C 180,E1 5418.735,E2 5418.735} C_VEL
LIN {X 0,Y 337.224,Z 362.849,A -85,B 0,C 180,E1 5417.348,E2 5417.348} C_VEL
LIN {X 0,Y 337.665,Z 356.354,A -85,B 0,C 180,E1 5417.112,E2 5417.112} C_VEL
LIN {X 0,Y 338.297,Z 349.512,A -85,B 0,C 180,E1 5416.97,E2 5416.97} C_VEL
LIN {X 0,Y 335.771,Z 343.804,A -85,B 0,C 180,E1 5414.662,E2 5414.662} C_VEL
LIN {X 0,Y 333.25,Z 338.137,A -85,B 0,C 180,E1 5411.773,E2 5411.773} C_VEL
LIN {X 0,Y 331.984,Z 335.295,A -85,B 0,C 180,E1 5409.885,E2 5409.885} C_VEL
LIN {X 0,Y 330.68,Z 332.15,A -85,B 0,C 180,E1 5407.122,E2 5407.122} C_VEL
LIN {X 0,Y 329.897,Z 329.512,A -85,B 0,C 180,E1 5402.085,E2 5402.085} C_VEL
LIN {X 0,Y 330.225,Z 330.007,A -85,B 0,C 180,E1 5399.653,E2 5399.653} C_VEL
LIN {X 0,Y 332.355,Z 333.243,A -85,B 0,C 180,E1 5394.822,E2 5394.822} C_VEL
LIN {X 0,Y 334.918,Z 337.934,A -85,B 0,C 180,E1 5391.502,E2 5391.502} C_VEL
LIN {X 0,Y 337.976,Z 343.622,A -85,B 0,C 180,E1 5388.568,E2 5388.568} C_VEL
LIN {X 0,Y 339.482,Z 346.907,A -85,B 0,C 180,E1 5387.301,E2 5387.301} C_VEL
LIN {X 0,Y 323.094,Z 511.762,A -85,B 0,C 180,E1 5384.127,E2 5384.127} C_VEL
LIN {X 0,Y 319.182,Z 534.928,A -85,B 0,C 180,E1 5383.561,E2 5383.561} C_VEL
LIN {X 0,Y 313.937,Z 557.483,A -85,B 0,C 180,E1 5382.832,E2 5382.832} C_VEL
LIN {X 0,Y 307.645,Z 578.511,A -85,B 0,C 180,E1 5381.917,E2 5381.917} C_VEL
LIN {X 0,Y 299.791,Z 600.212,A -85,B 0,C 180,E1 5380.705,E2 5380.705} C_VEL
LIN {X 0,Y 290.884,Z 621.167,A -85,B 0,C 180,E1 5379.215,E2 5379.215} C_VEL
LIN {X 0,Y 281.385,Z 640.258,A -85,B 0,C 180,E1 5377.495,E2 5377.495} C_VEL
LIN {X 0,Y 270.631,Z 659.547,A -85,B 0,C 180,E1 5375.325,E2 5375.325} C_VEL
LIN {X 0,Y 260.342,Z 676.093,A -85,B 0,C 180,E1 5372.997,E2 5372.997} C_VEL
LIN {X 0,Y 248.6,Z 693.287,A -85,B 0,C 180,E1 5369.964,E2 5369.964} C_VEL
LIN {X 0,Y 237.297,Z 708.698,A -85,B 0,C 180,E1 5366.538,E2 5366.538} C_VEL
LIN {X 0,Y 226.419,Z 722.44,A -85,B 0,C 180,E1 5362.641,E2 5362.641} C_VEL
LIN {X 0,Y 215.107,Z 736.217,A -85,B 0,C 180,E1 5357.65,E2 5357.65} C_VEL
LIN {X 0,Y 205.715,Z 747.532,A -85,B 0,C 180,E1 5352.373,E2 5352.373} C_VEL
LIN {X 0,Y 197.554,Z 757.427,A -85,B 0,C 180,E1 5346.309,E2 5346.309} C_VEL
LIN {X 0,Y 191.084,Z 765.944,A -85,B 0,C 180,E1 5339.462,E2 5339.462} C_VEL
LIN {X 0,Y 187.142,Z 772.031,A -85,B 0,C 180,E1 5332.955,E2 5332.955} C_VEL
LIN {X 0,Y 184.855,Z 776.652,A -85,B 0,C 180,E1 5326.012,E2 5326.012} C_VEL
LIN {X 0,Y 184.118,Z 779.24,A -85,B 0,C 180,E1 5320.323,E2 5320.323} C_VEL
LIN {X 0,Y 184.007,Z 780.826,A -85,B 0,C 180,E1 5314.363,E2 5314.363} C_VEL
LIN {X 0,Y 184.043,Z 781.099,A -85,B 0,C 180,E1 5309.066,E2 5309.066} C_VEL
LIN {X 0,Y 184.014,Z 780.4,A -85,B 0,C 180,E1 5303.761,E2 5303.761} C_VEL
LIN {X 0,Y 184.216,Z 778.738,A -85,B 0,C 180,E1 5298.415,E2 5298.415} C_VEL
LIN {X 0,Y 185.392,Z 775.387,A -85,B 0,C 180,E1 5291.772,E2 5291.772} C_VEL
LIN {X 0,Y 188.083,Z 770.391,A -85,B 0,C 180,E1 5285.168,E2 5285.168} C_VEL
LIN {X 0,Y 192.806,Z 763.55,A -85,B 0,C 180,E1 5278.416,E2 5278.416} C_VEL
LIN {X 0,Y 198.905,Z 755.684,A -85,B 0,C 180,E1 5272.539,E2 5272.539} C_VEL
LIN {X 0,Y 207.574,Z 745.157,A -85,B 0,C 180,E1 5266.465,E2 5266.465} C_VEL
LIN {X 0,Y 217.135,Z 733.769,A -85,B 0,C 180,E1 5261.361,E2 5261.361} C_VEL
LIN {X 0,Y 227.567,Z 720.897,A -85,B 0,C 180,E1 5256.906,E2 5256.906} C_VEL
LIN {X 0,Y 239.18,Z 705.997,A -85,B 0,C 180,E1 5252.836,E2 5252.836} C_VEL
LIN {X 0,Y 250.122,Z 691.015,A -85,B 0,C 180,E1 5249.608,E2 5249.608} C_VEL
LIN {X 0,Y 261.412,Z 674.217,A -85,B 0,C 180,E1 5246.738,E2 5246.738} C_VEL
LIN {X 0,Y 272.163,Z 656.8,A -85,B 0,C 180,E1 5244.347,E2 5244.347} C_VEL
LIN {X 0,Y 282.545,Z 637.765,A -85,B 0,C 180,E1 5242.277,E2 5242.277} C_VEL
LIN {X 0,Y 292.473,Z 617.216,A -85,B 0,C 180,E1 5240.499,E2 5240.499} C_VEL
LIN {X 0,Y 301.015,Z 596.818,A -85,B 0,C 180,E1 5239.096,E2 5239.096} C_VEL
LIN {X 0,Y 308.465,Z 575.468,A -85,B 0,C 180,E1 5237.95,E2 5237.95} C_VEL
LIN {X 0,Y 314.991,Z 552.696,A -85,B 0,C 180,E1 5237.005,E2 5237.005} C_VEL
LIN {X 0,Y 319.889,Z 530.631,A -85,B 0,C 180,E1 5236.33,E2 5236.33} C_VEL
LIN {X 0,Y 323.449,Z 507.345,A -85,B 0,C 180,E1 5235.791,E2 5235.791} C_VEL
LIN {X 0,Y 339.327,Z 346.52,A -85,B 0,C 180,E1 5232.689,E2 5232.689} C_VEL
LIN {X 0,Y 335.796,Z 339.699,A -85,B 0,C 180,E1 5229.598,E2 5229.598} C_VEL
LIN {X 0,Y 333.631,Z 335.82,A -85,B 0,C 180,E1 5227.231,E2 5227.231} C_VEL
LIN {X 0,Y 331.731,Z 332.389,A -85,B 0,C 180,E1 5224.494,E2 5224.494} C_VEL
LIN {X 0,Y 329.813,Z 329.176,A -85,B 0,C 180,E1 5219.131,E2 5219.131} C_VEL
LIN {X 0,Y 329.646,Z 329.533,A -85,B 0,C 180,E1 5216.87,E2 5216.87} C_VEL
LIN {X 0,Y 330.773,Z 332.673,A -85,B 0,C 180,E1 5212.007,E2 5212.007} C_VEL
LIN {X 0,Y 332.63,Z 336.956,A -85,B 0,C 180,E1 5208.733,E2 5208.733} C_VEL
LIN {X 0,Y 335.148,Z 342.543,A -85,B 0,C 180,E1 5205.707,E2 5205.707} C_VEL
LIN {X 0,Y 337.981,Z 349.024,A -85,B 0,C 180,E1 5203.058,E2 5203.058} C_VEL
LIN {X 0,Y 338.118,Z 349.793,A -85,B 0,C 180,E1 5202.907,E2 5202.907} C_VEL
LIN {X 0,Y 322.394,Z 514.167,A -85,B 0,C 180,E1 5199.869,E2 5199.869} C_VEL
LIN {X 0,Y 318.601,Z 536.633,A -85,B 0,C 180,E1 5199.336,E2 5199.336} C_VEL
LIN {X 0,Y 313.48,Z 558.547,A -85,B 0,C 180,E1 5198.641,E2 5198.641} C_VEL
LIN {X 0,Y 307.314,Z 579.1,A -85,B 0,C 180,E1 5197.76,E2 5197.76} C_VEL
LIN {X 0,Y 299.624,Z 600.092,A -85,B 0,C 180,E1 5196.586,E2 5196.586} C_VEL
LIN {X 0,Y 290.891,Z 620.3,A -85,B 0,C 180,E1 5195.149,E2 5195.149} C_VEL
LIN {X 0,Y 281.571,Z 638.717,A -85,B 0,C 180,E1 5193.486,E2 5193.486} C_VEL
LIN {X 0,Y 271.039,Z 657.113,A -85,B 0,C 180,E1 5191.396,E2 5191.396} C_VEL
LIN {X 0,Y 260.192,Z 674.092,A -85,B 0,C 180,E1 5188.972,E2 5188.972} C_VEL
LIN {X 0,Y 249.153,Z 689.497,A -85,B 0,C 180,E1 5186.168,E2 5186.168} C_VEL
LIN {X 0,Y 237.269,Z 704.764,A -85,B 0,C 180,E1 5182.64,E2 5182.64} C_VEL
LIN {X 0,Y 226.216,Z 718.008,A -85,B 0,C 180,E1 5178.709,E2 5178.709} C_VEL
LIN {X 0,Y 216.069,Z 729.34,A -85,B 0,C 180,E1 5174.325,E2 5174.325} C_VEL
LIN {X 0,Y 206.361,Z 739.905,A -85,B 0,C 180,E1 5169.039,E2 5169.039} C_VEL
LIN {X 0,Y 198.39,Z 748.577,A -85,B 0,C 180,E1 5163.321,E2 5163.321} C_VEL
LIN {X 0,Y 192.192,Z 755.455,A -85,B 0,C 180,E1 5157.175,E2 5157.175} C_VEL
LIN {X 0,Y 187.649,Z 761.106,A -85,B 0,C 180,E1 5150.263,E2 5150.263} C_VEL
LIN {X 0,Y 185.269,Z 764.728,A -85,B 0,C 180,E1 5143.736,E2 5143.736} C_VEL
LIN {X 0,Y 184.277,Z 766.895,A -85,B 0,C 180,E1 5137.169,E2 5137.169} C_VEL
LIN {X 0,Y 184.067,Z 767.653,A -85,B 0,C 180,E1 5131.813,E2 5131.813} C_VEL
LIN {X 0,Y 184.103,Z 767.534,A -85,B 0,C 180,E1 5126.263,E2 5126.263} C_VEL
LIN {X 0,Y 184.555,Z 766.175,A -85,B 0,C 180,E1 5120.017,E2 5120.017} C_VEL
LIN {X 0,Y 185.964,Z 763.586,A -85,B 0,C 180,E1 5113.765,E2 5113.765} C_VEL
LIN {X 0,Y 189.217,Z 759.083,A -85,B 0,C 180,E1 5106.846,E2 5106.846} C_VEL
LIN {X 0,Y 194.299,Z 753.17,A -85,B 0,C 180,E1 5100.396,E2 5100.396} C_VEL
LIN {X 0,Y 201.493,Z 745.221,A -85,B 0,C 180,E1 5094.16,E2 5094.16} C_VEL
LIN {X 0,Y 210.211,Z 735.811,A -85,B 0,C 180,E1 5088.614,E2 5088.614} C_VEL
LIN {X 0,Y 220.077,Z 725.064,A -85,B 0,C 180,E1 5083.751,E2 5083.751} C_VEL
LIN {X 0,Y 230.712,Z 712.806,A -85,B 0,C 180,E1 5079.521,E2 5079.521} C_VEL
LIN {X 0,Y 242.443,Z 698.419,A -85,B 0,C 180,E1 5075.666,E2 5075.666} C_VEL
LIN {X 0,Y 253.775,Z 683.439,A -85,B 0,C 180,E1 5072.529,E2 5072.529} C_VEL
LIN {X 0,Y 264.616,Z 667.531,A -85,B 0,C 180,E1 5069.919,E2 5069.919} C_VEL
LIN {X 0,Y 275.753,Z 649.417,A -85,B 0,C 180,E1 5067.562,E2 5067.562} C_VEL
LIN {X 0,Y 285.691,Z 631.276,A -85,B 0,C 180,E1 5065.688,E2 5065.688} C_VEL
LIN {X 0,Y 294.707,Z 612.161,A -85,B 0,C 180,E1 5064.131,E2 5064.131} C_VEL
LIN {X 0,Y 303.13,Z 591.477,A -85,B 0,C 180,E1 5062.796,E2 5062.796} C_VEL
LIN {X 0,Y 309.648,Z 572.36,A -85,B 0,C 180,E1 5061.826,E2 5061.826} C_VEL
LIN {X 0,Y 315.686,Z 550.472,A -85,B 0,C 180,E1 5060.978,E2 5060.978} C_VEL
LIN {X 0,Y 320.384,Z 528.412,A -85,B 0,C 180,E1 5060.351,E2 5060.351} C_VEL
LIN {X 0,Y 323.493,Z 506.016,A -85,B 0,C 180,E1 5059.868,E2 5059.868} C_VEL
LIN {X 0,Y 337.665,Z 356.354,A -85,B 0,C 180,E1 5057.112,E2 5057.112} C_VEL
LIN {X 0,Y 337.664,Z 354.032,A -85,B 0,C 180,E1 5056.923,E2 5056.923} C_VEL
LIN {X 0,Y 337.212,Z 352.045,A -85,B 0,C 180,E1 5056.458,E2 5056.458} C_VEL
LIN {X 0,Y 336.2,Z 350.71,A -85,B 0,C 180,E1 5055.632,E2 5055.632} C_VEL
LIN {X 0,Y 333.714,Z 349.633,A -85,B 0,C 180,E1 5053.557,E2 5053.557} C_VEL
LIN {X 0,Y 333.443,Z 349.174,A -85,B 0,C 180,E1 5053.268,E2 5053.268} C_VEL
LIN {X 0,Y 331.218,Z 343.78,A -85,B 0,C 180,E1 5050.238,E2 5050.238} C_VEL
LIN {X 0,Y 329.573,Z 339.928,A -85,B 0,C 180,E1 5046.795,E2 5046.795} C_VEL
LIN {X 0,Y 328.935,Z 337.424,A -85,B 0,C 180,E1 5041.916,E2 5041.916} C_VEL
LIN {X 0,Y 329.32,Z 338.144,A -85,B 0,C 180,E1 5039.304,E2 5039.304} C_VEL
LIN {X 0,Y 331.198,Z 341.041,A -85,B 0,C 180,E1 5035.064,E2 5035.064} C_VEL
LIN {X 0,Y 333.597,Z 345.615,A -85,B 0,C 180,E1 5031.815,E2 5031.815} C_VEL
LIN {X 0,Y 336.459,Z 351.167,A -85,B 0,C 180,E1 5028.95,E2 5028.95} C_VEL
LIN {X 0,Y 336.911,Z 352.508,A -85,B 0,C 180,E1 5028.513,E2 5028.513} C_VEL
LIN {X 0,Y 320.681,Z 511.967,A -85,B 0,C 180,E1 5025.486,E2 5025.486} C_VEL
LIN {X 0,Y 316.706,Z 535.018,A -85,B 0,C 180,E1 5024.936,E2 5024.936} C_VEL
LIN {X 0,Y 311.631,Z 556.631,A -85,B 0,C 180,E1 5024.263,E2 5024.263} C_VEL
LIN {X 0,Y 305.21,Z 577.771,A -85,B 0,C 180,E1 5023.374,E2 5023.374} C_VEL
LIN {X 0,Y 296.768,Z 600.64,A -85,B 0,C 180,E1 5022.131,E2 5022.131} C_VEL
LIN {X 0,Y 288.071,Z 620.638,A -85,B 0,C 180,E1 5020.743,E2 5020.743} C_VEL
LIN {X 0,Y 278.334,Z 639.801,A -85,B 0,C 180,E1 5019.063,E2 5019.063} C_VEL
LIN {X 0,Y 267.712,Z 658.46,A -85,B 0,C 180,E1 5017.022,E2 5017.022} C_VEL
LIN {X 0,Y 256.677,Z 675.705,A -85,B 0,C 180,E1 5014.65,E2 5014.65} C_VEL
LIN {X 0,Y 244.351,Z 693.169,A -85,B 0,C 180,E1 5011.61,E2 5011.61} C_VEL
LIN {X 0,Y 232.784,Z 708.36,A -85,B 0,C 180,E1 5008.258,E2 5008.258} C_VEL
LIN {X 0,Y 221.43,Z 722.108,A -85,B 0,C 180,E1 5004.367,E2 5004.367} C_VEL
LIN {X 0,Y 210.065,Z 735.305,A -85,B 0,C 180,E1 4999.6,E2 4999.6} C_VEL
LIN {X 0,Y 200.192,Z 746.505,A -85,B 0,C 180,E1 4994.364,E2 4994.364} C_VEL
LIN {X 0,Y 191.582,Z 756.271,A -85,B 0,C 180,E1 4988.392,E2 4988.392} C_VEL
LIN {X 0,Y 184.775,Z 764.529,A -85,B 0,C 180,E1 4981.837,E2 4981.837} C_VEL
LIN {X 0,Y 180.208,Z 770.679,A -85,B 0,C 180,E1 4975.261,E2 4975.261} C_VEL
LIN {X 0,Y 177.32,Z 775.67,A -85,B 0,C 180,E1 4968.067,E2 4968.067} C_VEL
LIN {X 0,Y 176.232,Z 778.579,A -85,B 0,C 180,E1 4961.785,E2 4961.785} C_VEL
LIN {X 0,Y 176.01,Z 780.262,A -85,B 0,C 180,E1 4955.869,E2 4955.869} C_VEL
LIN {X 0,Y 176.056,Z 780.873,A -85,B 0,C 180,E1 4950,E2 4950} C_VEL
LIN {X 0,Y 176.012,Z 780.253,A -85,B 0,C 180,E1 4944.131,E2 4944.131} C_VEL
LIN {X 0,Y 176.202,Z 778.687,A -85,B 0,C 180,E1 4938.545,E2 4938.545} C_VEL
LIN {X 0,Y 177.232,Z 775.821,A -85,B 0,C 180,E1 4932.264,E2 4932.264} C_VEL
LIN {X 0,Y 180.049,Z 770.892,A -85,B 0,C 180,E1 4925.037,E2 4925.037} C_VEL
LIN {X 0,Y 184.643,Z 764.644,A -85,B 0,C 180,E1 4918.315,E2 4918.315} C_VEL
LIN {X 0,Y 191.215,Z 756.639,A -85,B 0,C 180,E1 4911.903,E2 4911.903} C_VEL
LIN {X 0,Y 199.734,Z 746.971,A -85,B 0,C 180,E1 4905.909,E2 4905.909} C_VEL
LIN {X 0,Y 209.527,Z 735.817,A -85,B 0,C 180,E1 4900.648,E2 4900.648} C_VEL
LIN {X 0,Y 220.819,Z 722.724,A -85,B 0,C 180,E1 4895.857,E2 4895.857} C_VEL
LIN {X 0,Y 232.115,Z 709.034,A -85,B 0,C 180,E1 4891.943,E2 4891.943} C_VEL
LIN {X 0,Y 243.986,Z 693.493,A -85,B 0,C 180,E1 4888.478,E2 4888.478} C_VEL
LIN {X 0,Y 255.919,Z 676.655,A -85,B 0,C 180,E1 4885.515,E2 4885.515} C_VEL
LIN {X 0,Y 266.871,Z 659.566,A -85,B 0,C 180,E1 4883.136,E2 4883.136} C_VEL
LIN {X 0,Y 277.519,Z 641.032,A -85,B 0,C 180,E1 4881.075,E2 4881.075} C_VEL
LIN {X 0,Y 287.647,Z 621.219,A -85,B 0,C 180,E1 4879.316,E2 4879.316} C_VEL
LIN {X 0,Y 296.334,Z 601.304,A -85,B 0,C 180,E1 4877.924,E2 4877.924} C_VEL
LIN {X 0,Y 304.413,Z 579.698,A -85,B 0,C 180,E1 4876.729,E2 4876.729} C_VEL
LIN {X 0,Y 310.958,Z 558.371,A -85,B 0,C 180,E1 4875.816,E2 4875.816} C_VEL
LIN {X 0,Y 316.421,Z 535.576,A -85,B 0,C 180,E1 4875.09,E2 4875.09} C_VEL
LIN {X 0,Y 320.438,Z 512.535,A -85,B 0,C 180,E1 4874.535,E2 4874.535} C_VEL
LIN {X 0,Y 332.749,Z 391.849,A -85,B 0,C 180,E1 4872.232,E2 4872.232} C_VEL
LIN {X 0,Y 336.757,Z 352.058,A -85,B 0,C 180,E1 4871.474,E2 4871.474} C_VEL
LIN {X 0,Y 333.874,Z 346.352,A -85,B 0,C 180,E1 4868.698,E2 4868.698} C_VEL
LIN {X 0,Y 332.151,Z 343.167,A -85,B 0,C 180,E1 4866.655,E2 4866.655} C_VEL
LIN {X 0,Y 330.639,Z 340.261,A -85,B 0,C 180,E1 4864.335,E2 4864.335} C_VEL
LIN {X 0,Y 328.81,Z 337.075,A -85,B 0,C 180,E1 4858.954,E2 4858.954} C_VEL
LIN {X 0,Y 328.672,Z 337.597,A -85,B 0,C 180,E1 4856.686,E2 4856.686} C_VEL
LIN {X 0,Y 329.721,Z 340.603,A -85,B 0,C 180,E1 4852.157,E2 4852.157} C_VEL
LIN {X 0,Y 331.41,Z 344.661,A -85,B 0,C 180,E1 4849.043,E2 4849.043} C_VEL
LIN {X 0,Y 333.792,Z 350.22,A -85,B 0,C 180,E1 4846.048,E2 4846.048} C_VEL
LIN {X 0,Y 335.686,Z 354.778,A -85,B 0,C 180,E1 4844.142,E2 4844.142} C_VEL
LIN {X 0,Y 320.02,Z 514.111,A -85,B 0,C 180,E1 4841.236,E2 4841.236} C_VEL
LIN {X 0,Y 316.128,Z 536.695,A -85,B 0,C 180,E1 4840.714,E2 4840.714} C_VEL
LIN {X 0,Y 310.884,Z 558.669,A -85,B 0,C 180,E1 4840.035,E2 4840.035} C_VEL
LIN {X 0,Y 304.387,Z 579.84,A -85,B 0,C 180,E1 4839.148,E2 4839.148} C_VEL
LIN {X 0,Y 296.539,Z 600.678,A -85,B 0,C 180,E1 4838.004,E2 4838.004} C_VEL
LIN {X 0,Y 288.057,Z 619.905,A -85,B 0,C 180,E1 4836.67,E2 4836.67} C_VEL
LIN {X 0,Y 278.413,Z 638.542,A -85,B 0,C 180,E1 4835.031,E2 4835.031} C_VEL
LIN {X 0,Y 267.267,Z 657.512,A -85,B 0,C 180,E1 4832.916,E2 4832.916} C_VEL
LIN {X 0,Y 256.11,Z 674.463,A -85,B 0,C 180,E1 4830.525,E2 4830.525} C_VEL
LIN {X 0,Y 244.722,Z 689.846,A -85,B 0,C 180,E1 4827.748,E2 4827.748} C_VEL
LIN {X 0,Y 232.658,Z 704.811,A -85,B 0,C 180,E1 4824.313,E2 4824.313} C_VEL
LIN {X 0,Y 221.156,Z 718.047,A -85,B 0,C 180,E1 4820.396,E2 4820.396} C_VEL
LIN {X 0,Y 210.288,Z 729.652,A -85,B 0,C 180,E1 4815.885,E2 4815.885} C_VEL
LIN {X 0,Y 199.615,Z 740.654,A -85,B 0,C 180,E1 4810.251,E2 4810.251} C_VEL
LIN {X 0,Y 191.239,Z 749.257,A -85,B 0,C 180,E1 4804.377,E2 4804.377} C_VEL
LIN {X 0,Y 184.485,Z 756.276,A -85,B 0,C 180,E1 4797.78,E2 4797.78} C_VEL
LIN {X 0,Y 179.704,Z 761.793,A -85,B 0,C 180,E1 4790.519,E2 4790.519} C_VEL
LIN {X 0,Y 177.254,Z 765.325,A -85,B 0,C 180,E1 4783.704,E2 4783.704} C_VEL
LIN {X 0,Y 176.264,Z 767.297,A -85,B 0,C 180,E1 4776.928,E2 4776.928} C_VEL
LIN {X 0,Y 176.071,Z 767.983,A -85,B 0,C 180,E1 4771.302,E2 4771.302} C_VEL
LIN {X 0,Y 176.136,Z 767.78,A -85,B 0,C 180,E1 4765.442,E2 4765.442} C_VEL
LIN {X 0,Y 176.717,Z 766.255,A -85,B 0,C 180,E1 4758.909,E2 4758.909} C_VEL
LIN {X 0,Y 178.543,Z 763.428,A -85,B 0,C 180,E1 4752.061,E2 4752.061} C_VEL
LIN {X 0,Y 182.284,Z 758.753,A -85,B 0,C 180,E1 4745.017,E2 4745.017} C_VEL
LIN {X 0,Y 188.457,Z 752.113,A -85,B 0,C 180,E1 4737.958,E2 4737.958} C_VEL
LIN {X 0,Y 196.118,Z 744.349,A -85,B 0,C 180,E1 4731.912,E2 4731.912} C_VEL
LIN {X 0,Y 205.595,Z 734.62,A -85,B 0,C 180,E1 4726.325,E2 4726.325} C_VEL
LIN {X 0,Y 216.734,Z 722.906,A -85,B 0,C 180,E1 4721.241,E2 4721.241} C_VEL
LIN {X 0,Y 228.089,Z 710.369,A -85,B 0,C 180,E1 4717.08,E2 4717.08} C_VEL
LIN {X 0,Y 239.798,Z 696.27,A -85,B 0,C 180,E1 4713.499,E2 4713.499} C_VEL
LIN {X 0,Y 251.998,Z 680.313,A -85,B 0,C 180,E1 4710.35,E2 4710.35} C_VEL
LIN {X 0,Y 263.379,Z 663.939,A -85,B 0,C 180,E1 4707.809,E2 4707.809} C_VEL
LIN {X 0,Y 274.054,Z 646.54,A -85,B 0,C 180,E1 4705.693,E2 4705.693} C_VEL
LIN {X 0,Y 284.511,Z 627.322,A -85,B 0,C 180,E1 4703.838,E2 4703.838} C_VEL
LIN {X 0,Y 293.565,Z 608.226,A -85,B 0,C 180,E1 4702.38,E2 4702.38} C_VEL
LIN {X 0,Y 301.492,Z 588.414,A -85,B 0,C 180,E1 4701.192,E2 4701.192} C_VEL
LIN {X 0,Y 308.357,Z 568.148,A -85,B 0,C 180,E1 4700.234,E2 4700.234} C_VEL
LIN {X 0,Y 313.883,Z 547.592,A -85,B 0,C 180,E1 4699.499,E2 4699.499} C_VEL
LIN {X 0,Y 318.686,Z 523.922,A -85,B 0,C 180,E1 4698.879,E2 4698.879} C_VEL
LIN {X 0,Y 321.705,Z 500.974,A -85,B 0,C 180,E1 4698.408,E2 4698.408} C_VEL
LIN {X 0,Y 335.819,Z 354.719,A -85,B 0,C 180,E1 4695.721,E2 4695.721} C_VEL
LIN {X 0,Y 333.443,Z 349.174,A -85,B 0,C 180,E1 4693.268,E2 4693.268} C_VEL
LIN {X 0,Y 332.255,Z 347.81,A -85,B 0,C 180,E1 4691.97,E2 4691.97} C_VEL
LIN {X 0,Y 330.238,Z 348.259,A -85,B 0,C 180,E1 4689.672,E2 4689.672} C_VEL
LIN {X 0,Y 328.925,Z 348.492,A -85,B 0,C 180,E1 4687.628,E2 4687.628} C_VEL
LIN {X 0,Y 328.724,Z 348.161,A -85,B 0,C 180,E1 4687.142,E2 4687.142} C_VEL
LIN {X 0,Y 327.955,Z 345.372,A -85,B 0,C 180,E1 4681.922,E2 4681.922} C_VEL
LIN {X 0,Y 328.337,Z 346.116,A -85,B 0,C 180,E1 4679.302,E2 4679.302} C_VEL
LIN {X 0,Y 330.096,Z 348.959,A -85,B 0,C 180,E1 4675.222,E2 4675.222} C_VEL
LIN {X 0,Y 332.353,Z 353.448,A -85,B 0,C 180,E1 4672.046,E2 4672.046} C_VEL
LIN {X 0,Y 334.513,Z 357.877,A -85,B 0,C 180,E1 4669.748,E2 4669.748} C_VEL
LIN {X 0,Y 318.464,Z 512.065,A -85,B 0,C 180,E1 4666.867,E2 4666.867} C_VEL
LIN {X 0,Y 314.415,Z 535.116,A -85,B 0,C 180,E1 4666.332,E2 4666.332} C_VEL
LIN {X 0,Y 309.195,Z 556.889,A -85,B 0,C 180,E1 4665.672,E2 4665.672} C_VEL
LIN {X 0,Y 302.543,Z 578.331,A -85,B 0,C 180,E1 4664.794,E2 4664.794} C_VEL
LIN {X 0,Y 294.107,Z 600.657,A -85,B 0,C 180,E1 4663.611,E2 4663.611} C_VEL
LIN {X 0,Y 285.041,Z 621.027,A -85,B 0,C 180,E1 4662.232,E2 4662.232} C_VEL
LIN {X 0,Y 274.676,Z 640.836,A -85,B 0,C 180,E1 4660.522,E2 4660.522} C_VEL
LIN {X 0,Y 262.942,Z 660.619,A -85,B 0,C 180,E1 4658.356,E2 4658.356} C_VEL
LIN {X 0,Y 251.407,Z 678.023,A -85,B 0,C 180,E1 4655.944,E2 4655.944} C_VEL
LIN {X 0,Y 239.045,Z 694.705,A -85,B 0,C 180,E1 4652.986,E2 4652.986} C_VEL
LIN {X 0,Y 226.45,Z 710.4,A -85,B 0,C 180,E1 4649.426,E2 4649.426} C_VEL
LIN {X 0,Y 214.776,Z 723.938,A -85,B 0,C 180,E1 4645.485,E2 4645.485} C_VEL
LIN {X 0,Y 203.053,Z 736.761,A -85,B 0,C 180,E1 4640.63,E2 4640.63} C_VEL
LIN {X 0,Y 192.518,Z 748.053,A -85,B 0,C 180,E1 4635.064,E2 4635.064} C_VEL
LIN {X 0,Y 183.929,Z 757.229,A -85,B 0,C 180,E1 4629.092,E2 4629.092} C_VEL
LIN {X 0,Y 176.474,Z 765.653,A -85,B 0,C 180,E1 4621.796,E2 4621.796} C_VEL
LIN {X 0,Y 171.661,Z 771.954,A -85,B 0,C 180,E1 4614.427,E2 4614.427} C_VEL
LIN {X 0,Y 169.074,Z 776.227,A -85,B 0,C 180,E1 4607.198,E2 4607.198} C_VEL
LIN {X 0,Y 168.114,Z 779.016,A -85,B 0,C 180,E1 4600.278,E2 4600.278} C_VEL
LIN {X 0,Y 168.019,Z 780.296,A -85,B 0,C 180,E1 4594.095,E2 4594.095} C_VEL
LIN {X 0,Y 168.05,Z 780.493,A -85,B 0,C 180,E1 4588.636,E2 4588.636} C_VEL
LIN {X 0,Y 168.03,Z 779.814,A -85,B 0,C 180,E1 4583.165,E2 4583.165} C_VEL
LIN {X 0,Y 168.36,Z 778.024,A -85,B 0,C 180,E1 4576.958,E2 4576.958} C_VEL
LIN {X 0,Y 170.077,Z 774.346,A -85,B 0,C 180,E1 4569.346,E2 4569.346} C_VEL
LIN {X 0,Y 173.355,Z 769.514,A -85,B 0,C 180,E1 4562.522,E2 4562.522} C_VEL
LIN {X 0,Y 179.412,Z 762.192,A -85,B 0,C 180,E1 4554.97,E2 4554.97} C_VEL
LIN {X 0,Y 187.267,Z 753.619,A -85,B 0,C 180,E1 4548.373,E2 4548.373} C_VEL
LIN {X 0,Y 196.725,Z 743.451,A -85,B 0,C 180,E1 4542.528,E2 4542.528} C_VEL
LIN {X 0,Y 207.569,Z 731.816,A -85,B 0,C 180,E1 4537.366,E2 4537.366} C_VEL
LIN {X 0,Y 218.538,Z 719.507,A -85,B 0,C 180,E1 4533.15,E2 4533.15} C_VEL
LIN {X 0,Y 231.228,Z 704.426,A -85,B 0,C 180,E1 4529.138,E2 4529.138} C_VEL
LIN {X 0,Y 243.434,Z 688.866,A -85,B 0,C 180,E1 4525.911,E2 4525.911} C_VEL
LIN {X 0,Y 255.148,Z 672.299,A -85,B 0,C 180,E1 4523.232,E2 4523.232} C_VEL
LIN {X 0,Y 266.569,Z 654.569,A -85,B 0,C 180,E1 4520.943,E2 4520.943} C_VEL
LIN {X 0,Y 276.72,Z 636.836,A -85,B 0,C 180,E1 4519.12,E2 4519.12} C_VEL
LIN {X 0,Y 287.137,Z 616.126,A -85,B 0,C 180,E1 4517.43,E2 4517.43} C_VEL
LIN {X 0,Y 295.639,Z 596.638,A -85,B 0,C 180,E1 4516.164,E2 4516.164} C_VEL
LIN {X 0,Y 303.276,Z 575.622,A -85,B 0,C 180,E1 4515.097,E2 4515.097} C_VEL
LIN {X 0,Y 309.987,Z 553.175,A -85,B 0,C 180,E1 4514.213,E2 4514.213} C_VEL
LIN {X 0,Y 315.059,Z 531.205,A -85,B 0,C 180,E1 4513.576,E2 4513.576} C_VEL
LIN {X 0,Y 318.805,Z 507.813,A -85,B 0,C 180,E1 4513.057,E2 4513.057} C_VEL
LIN {X 0,Y 334.348,Z 357.67,A -85,B 0,C 180,E1 4510.249,E2 4510.249} C_VEL
LIN {X 0,Y 331.561,Z 351.945,A -85,B 0,C 180,E1 4507.189,E2 4507.189} C_VEL
LIN {X 0,Y 329.46,Z 347.997,A -85,B 0,C 180,E1 4504.002,E2 4504.002} C_VEL
LIN {X 0,Y 327.812,Z 344.977,A -85,B 0,C 180,E1 4498.776,E2 4498.776} C_VEL
LIN {X 0,Y 327.738,Z 345.941,A -85,B 0,C 180,E1 4495.976,E2 4495.976} C_VEL
LIN {X 0,Y 328.635,Z 348.417,A -85,B 0,C 180,E1 4492.395,E2 4492.395} C_VEL
LIN {X 0,Y 330.206,Z 352.366,A -85,B 0,C 180,E1 4489.356,E2 4489.356} C_VEL
LIN {X 0,Y 332.417,Z 357.803,A -85,B 0,C 180,E1 4486.431,E2 4486.431} C_VEL
LIN {X 0,Y 333.349,Z 360.4,A -85,B 0,C 180,E1 4485.384,E2 4485.384} C_VEL
LIN {X 0,Y 317.833,Z 514.034,A -85,B 0,C 180,E1 4482.623,E2 4482.623} C_VEL
LIN {X 0,Y 313.867,Z 536.623,A -85,B 0,C 180,E1 4482.115,E2 4482.115} C_VEL
LIN {X 0,Y 308.473,Z 558.792,A -85,B 0,C 180,E1 4481.452,E2 4481.452} C_VEL
LIN {X 0,Y 302.065,Z 579.306,A -85,B 0,C 180,E1 4480.621,E2 4480.621} C_VEL
LIN {X 0,Y 294.056,Z 600.268,A -85,B 0,C 180,E1 4479.51,E2 4479.51} C_VEL
LIN {X 0,Y 285.205,Z 619.949,A -85,B 0,C 180,E1 4478.185,E2 4478.185} C_VEL
LIN {X 0,Y 275.569,Z 638.171,A -85,B 0,C 180,E1 4476.627,E2 4476.627} C_VEL
LIN {X 0,Y 264.029,Z 657.39,A -85,B 0,C 180,E1 4474.543,E2 4474.543} C_VEL
LIN {X 0,Y 252.598,Z 674.313,A -85,B 0,C 180,E1 4472.209,E2 4472.209} C_VEL
LIN {X 0,Y 240.484,Z 690.198,A -85,B 0,C 180,E1 4469.386,E2 4469.386} C_VEL
LIN {X 0,Y 228.001,Z 705.139,A -85,B 0,C 180,E1 4465.976,E2 4465.976} C_VEL
LIN {X 0,Y 216.393,Z 717.977,A -85,B 0,C 180,E1 4462.194,E2 4462.194} C_VEL
LIN {X 0,Y 205.099,Z 729.537,A -85,B 0,C 180,E1 4457.72,E2 4457.72} C_VEL
LIN {X 0,Y 194.375,Z 740.071,A -85,B 0,C 180,E1 4452.364,E2 4452.364} C_VEL
LIN {X 0,Y 185.294,Z 748.796,A -85,B 0,C 180,E1 4446.409,E2 4446.409} C_VEL
LIN {X 0,Y 177.855,Z 755.995,A -85,B 0,C 180,E1 4439.65,E2 4439.65} C_VEL
LIN {X 0,Y 172.457,Z 761.699,A -85,B 0,C 180,E1 4432.138,E2 4432.138} C_VEL
LIN {X 0,Y 169.578,Z 765.318,A -85,B 0,C 180,E1 4425.036,E2 4425.036} C_VEL
LIN {X 0,Y 168.342,Z 767.48,A -85,B 0,C 180,E1 4417.851,E2 4417.851} C_VEL
LIN {X 0,Y 168.08,Z 768.234,A -85,B 0,C 180,E1 4412.003,E2 4412.003} C_VEL
LIN {X 0,Y 168.113,Z 768.137,A -85,B 0,C 180,E1 4406.249,E2 4406.249} C_VEL
LIN {X 0,Y 168.64,Z 766.868,A -85,B 0,C 180,E1 4399.409,E2 4399.409} C_VEL
LIN {X 0,Y 170.307,Z 764.326,A -85,B 0,C 180,E1 4392.578,E2 4392.578} C_VEL
LIN {X 0,Y 174.226,Z 759.777,A -85,B 0,C 180,E1 4384.871,E2 4384.871} C_VEL
LIN {X 0,Y 180.237,Z 753.771,A -85,B 0,C 180,E1 4377.823,E2 4377.823} C_VEL
LIN {X 0,Y 188.376,Z 745.884,A -85,B 0,C 180,E1 4371.284,E2 4371.284} C_VEL
LIN {X 0,Y 198.209,Z 736.424,A -85,B 0,C 180,E1 4365.48,E2 4365.48} C_VEL
LIN {X 0,Y 209.092,Z 725.693,A -85,B 0,C 180,E1 4360.509,E2 4360.509} C_VEL
LIN {X 0,Y 220.679,Z 713.443,A -85,B 0,C 180,E1 4356.248,E2 4356.248} C_VEL
LIN {X 0,Y 233.524,Z 698.844,A -85,B 0,C 180,E1 4352.358,E2 4352.358} C_VEL
LIN {X 0,Y 245.43,Z 684.152,A -85,B 0,C 180,E1 4349.333,E2 4349.333} C_VEL
LIN {X 0,Y 257.013,Z 668.155,A -85,B 0,C 180,E1 4346.773,E2 4346.773} C_VEL
LIN {X 0,Y 269.072,Z 649.588,A -85,B 0,C 180,E1 4344.442,E2 4344.442} C_VEL
LIN {X 0,Y 279.509,Z 631.432,A -85,B 0,C 180,E1 4342.648,E2 4342.648} C_VEL
LIN {X 0,Y 288.944,Z 612.309,A -85,B 0,C 180,E1 4341.164,E2 4341.164} C_VEL
LIN {X 0,Y 297.729,Z 591.632,A -85,B 0,C 180,E1 4339.899,E2 4339.899} C_VEL
LIN {X 0,Y 304.513,Z 572.535,A -85,B 0,C 180,E1 4338.984,E2 4338.984} C_VEL
LIN {X 0,Y 310.817,Z 550.591,A -85,B 0,C 180,E1 4338.181,E2 4338.181} C_VEL
LIN {X 0,Y 315.707,Z 528.531,A -85,B 0,C 180,E1 4337.588,E2 4337.588} C_VEL
LIN {X 0,Y 318.981,Z 505.97,A -85,B 0,C 180,E1 4337.122,E2 4337.122} C_VEL
LIN {X 0,Y 333.52,Z 360.26,A -85,B 0,C 180,E1 4334.497,E2 4334.497} C_VEL
LIN {X 0,Y 331.036,Z 354.083,A -85,B 0,C 180,E1 4331.499,E2 4331.499} C_VEL
LIN {X 0,Y 329.638,Z 350.715,A -85,B 0,C 180,E1 4329.251,E2 4329.251} C_VEL
LIN {X 0,Y 328.724,Z 348.161,A -85,B 0,C 180,E1 4327.142,E2 4327.142} C_VEL
LIN {X 0,Y 328.197,Z 348.003,A -85,B 0,C 180,E1 4325.796,E2 4325.796} C_VEL
LIN {X 0,Y 327.416,Z 350.4,A -85,B 0,C 180,E1 4323.691,E2 4323.691} C_VEL
LIN {X 0,Y 327.039,Z 353.109,A -85,B 0,C 180,E1 4321.467,E2 4321.467} C_VEL
LIN {X 0,Y 327.069,Z 353.344,A -85,B 0,C 180,E1 4320.975,E2 4320.975} C_VEL
LIN {X 0,Y 328.821,Z 356.399,A -85,B 0,C 180,E1 4315.728,E2 4315.728} C_VEL
LIN {X 0,Y 331.046,Z 361.129,A -85,B 0,C 180,E1 4312.363,E2 4312.363} C_VEL
LIN {X 0,Y 332.222,Z 363.737,A -85,B 0,C 180,E1 4310.99,E2 4310.99} C_VEL
LIN {X 0,Y 316.448,Z 512.047,A -85,B 0,C 180,E1 4308.269,E2 4308.269} C_VEL
LIN {X 0,Y 312.341,Z 535.083,A -85,B 0,C 180,E1 4307.75,E2 4307.75} C_VEL
LIN {X 0,Y 306.943,Z 557.167,A -85,B 0,C 180,E1 4307.102,E2 4307.102} C_VEL
LIN {X 0,Y 300.065,Z 578.891,A -85,B 0,C 180,E1 4306.238,E2 4306.238} C_VEL
LIN {X 0,Y 291.469,Z 601.087,A -85,B 0,C 180,E1 4305.092,E2 4305.092} C_VEL
LIN {X 0,Y 282.151,Z 621.505,A -85,B 0,C 180,E1 4303.743,E2 4303.743} C_VEL
LIN {X 0,Y 271.631,Z 641.11,A -85,B 0,C 180,E1 4302.09,E2 4302.09} C_VEL
LIN {X 0,Y 259.643,Z 660.765,A -85,B 0,C 180,E1 4299.983,E2 4299.983} C_VEL
LIN {X 0,Y 247.658,Z 678.322,A -85,B 0,C 180,E1 4297.594,E2 4297.594} C_VEL
LIN {X 0,Y 234.966,Z 694.863,A -85,B 0,C 180,E1 4294.696,E2 4294.696} C_VEL
LIN {X 0,Y 221.605,Z 710.853,A -85,B 0,C 180,E1 4291.078,E2 4291.078} C_VEL
LIN {X 0,Y 208.937,Z 724.944,A -85,B 0,C 180,E1 4286.939,E2 4286.939} C_VEL
LIN {X 0,Y 196.874,Z 737.424,A -85,B 0,C 180,E1 4282.084,E2 4282.084} C_VEL
LIN {X 0,Y 185.055,Z 749.316,A -85,B 0,C 180,E1 4275.938,E2 4275.938} C_VEL
LIN {X 0,Y 175.918,Z 758.601,A -85,B 0,C 180,E1 4269.535,E2 4269.535} C_VEL
LIN {X 0,Y 168.577,Z 766.304,A -85,B 0,C 180,E1 4262.262,E2 4262.262} C_VEL
LIN {X 0,Y 163.448,Z 772.539,A -85,B 0,C 180,E1 4254.195,E2 4254.195} C_VEL
LIN {X 0,Y 160.999,Z 776.44,A -85,B 0,C 180,E1 4246.97,E2 4246.97} C_VEL
LIN {X 0,Y 160.071,Z 779.084,A -85,B 0,C 180,E1 4239.346,E2 4239.346} C_VEL
LIN {X 0,Y 160.034,Z 780.081,A -85,B 0,C 180,E1 4233.223,E2 4233.223} C_VEL
LIN {X 0,Y 160.049,Z 780.178,A -85,B 0,C 180,E1 4228.21,E2 4228.21} C_VEL
LIN {X 0,Y 160.04,Z 779.447,A -85,B 0,C 180,E1 4222.461,E2 4222.461} C_VEL
LIN {X 0,Y 160.482,Z 777.605,A -85,B 0,C 180,E1 4215.938,E2 4215.938} C_VEL
LIN {X 0,Y 162.522,Z 773.826,A -85,B 0,C 180,E1 4207.959,E2 4207.959} C_VEL
LIN {X 0,Y 166.263,Z 768.941,A -85,B 0,C 180,E1 4200.85,E2 4200.85} C_VEL
LIN {X 0,Y 172.625,Z 761.881,A -85,B 0,C 180,E1 4193.376,E2 4193.376} C_VEL
LIN {X 0,Y 180.892,Z 753.485,A -85,B 0,C 180,E1 4186.735,E2 4186.735} C_VEL
LIN {X 0,Y 191.144,Z 743.132,A -85,B 0,C 180,E1 4180.671,E2 4180.671} C_VEL
LIN {X 0,Y 202.578,Z 731.487,A -85,B 0,C 180,E1 4175.476,E2 4175.476} C_VEL
LIN {X 0,Y 214.317,Z 718.905,A -85,B 0,C 180,E1 4171.188,E2 4171.188} C_VEL
LIN {X 0,Y 227.278,Z 704.075,A -85,B 0,C 180,E1 4167.299,E2 4167.299} C_VEL
LIN {X 0,Y 240.054,Z 688.311,A -85,B 0,C 180,E1 4164.09,E2 4164.09} C_VEL
LIN {X 0,Y 251.989,Z 671.909,A -85,B 0,C 180,E1 4161.497,E2 4161.497} C_VEL
LIN {X 0,Y 264.546,Z 652.775,A -85,B 0,C 180,E1 4159.117,E2 4159.117} C_VEL
LIN {X 0,Y 275.122,Z 634.633,A -85,B 0,C 180,E1 4157.338,E2 4157.338} C_VEL
LIN {X 0,Y 284.787,Z 615.582,A -85,B 0,C 180,E1 4155.855,E2 4155.855} C_VEL
LIN {X 0,Y 293.469,Z 596.037,A -85,B 0,C 180,E1 4154.632,E2 4154.632} C_VEL
LIN {X 0,Y 301.129,Z 575.238,A -85,B 0,C 180,E1 4153.615,E2 4153.615} C_VEL
LIN {X 0,Y 308.05,Z 552.309,A -85,B 0,C 180,E1 4152.751,E2 4152.751} C_VEL
LIN {X 0,Y 313.203,Z 530.195,A -85,B 0,C 180,E1 4152.138,E2 4152.138} C_VEL
LIN {X 0,Y 316.882,Z 507.096,A -85,B 0,C 180,E1 4151.643,E2 4151.643} C_VEL
LIN {X 0,Y 332.075,Z 363.437,A -85,B 0,C 180,E1 4149.008,E2 4149.008} C_VEL
LIN {X 0,Y 329.892,Z 358.977,A -85,B 0,C 180,E1 4146.351,E2 4146.351} C_VEL
LIN {X 0,Y 328.376,Z 355.869,A -85,B 0,C 180,E1 4143.841,E2 4143.841} C_VEL
LIN {X 0,Y 326.836,Z 352.924,A -85,B 0,C 180,E1 4138.773,E2 4138.773} C_VEL
LIN {X 0,Y 326.747,Z 353.825,A -85,B 0,C 180,E1 4136.14,E2 4136.14} C_VEL
LIN {X 0,Y 327.553,Z 356.23,A -85,B 0,C 180,E1 4132.634,E2 4132.634} C_VEL
LIN {X 0,Y 329.055,Z 360.215,A -85,B 0,C 180,E1 4129.584,E2 4129.584} C_VEL
LIN {X 0,Y 331.162,Z 365.68,A -85,B 0,C 180,E1 4126.69,E2 4126.69} C_VEL
LIN {X 0,Y 316.715,Z 506.749,A -85,B 0,C 180,E1 4124.166,E2 4124.166} C_VEL
LIN {X 0,Y 313.267,Z 529.618,A -85,B 0,C 180,E1 4123.701,E2 4123.701} C_VEL
LIN {X 0,Y 308.194,Z 551.765,A -85,B 0,C 180,E1 4123.117,E2 4123.117} C_VEL
LIN {X 0,Y 301.689,Z 573.667,A -85,B 0,C 180,E1 4122.328,E2 4122.328} C_VEL
LIN {X 0,Y 294.358,Z 593.759,A -85,B 0,C 180,E1 4121.379,E2 4121.379} C_VEL
LIN {X 0,Y 285.538,Z 613.743,A -85,B 0,C 180,E1 4120.165,E2 4120.165} C_VEL
LIN {X 0,Y 275.791,Z 632.818,A -85,B 0,C 180,E1 4118.702,E2 4118.702} C_VEL
LIN {X 0,Y 265.55,Z 650.195,A -85,B 0,C 180,E1 4117.01,E2 4117.01} C_VEL
LIN {X 0,Y 253.52,Z 668.236,A -85,B 0,C 180,E1 4114.789,E2 4114.789} C_VEL
LIN {X 0,Y 241.678,Z 684.159,A -85,B 0,C 180,E1 4112.292,E2 4112.292} C_VEL
LIN {X 0,Y 229.176,Z 699.122,A -85,B 0,C 180,E1 4109.255,E2 4109.255} C_VEL
LIN {X 0,Y 216.064,Z 713.507,A -85,B 0,C 180,E1 4105.456,E2 4105.456} C_VEL
LIN {X 0,Y 203.982,Z 725.784,A -85,B 0,C 180,E1 4101.201,E2 4101.201} C_VEL
LIN {X 0,Y 192.553,Z 736.544,A -85,B 0,C 180,E1 4096.2,E2 4096.2} C_VEL
LIN {X 0,Y 181.761,Z 746.364,A -85,B 0,C 180,E1 4090.06,E2 4090.06} C_VEL
LIN {X 0,Y 173.432,Z 753.939,A -85,B 0,C 180,E1 4083.603,E2 4083.603} C_VEL
LIN {X 0,Y 166.919,Z 759.977,A -85,B 0,C 180,E1 4076.312,E2 4076.312} C_VEL
LIN {X 0,Y 162.605,Z 764.559,A -85,B 0,C 180,E1 4068.276,E2 4068.276} C_VEL
LIN {X 0,Y 160.733,Z 767.117,A -85,B 0,C 180,E1 4061.118,E2 4061.118} C_VEL
LIN {X 0,Y 160.125,Z 768.419,A -85,B 0,C 180,E1 4053.938,E2 4053.938} C_VEL
LIN {X 0,Y 160.088,Z 768.531,A -85,B 0,C 180,E1 4047.852,E2 4047.852} C_VEL
LIN {X 0,Y 160.37,Z 767.798,A -85,B 0,C 180,E1 4041.756,E2 4041.756} C_VEL
LIN {X 0,Y 161.745,Z 765.675,A -85,B 0,C 180,E1 4034.217,E2 4034.217} C_VEL
LIN {X 0,Y 164.894,Z 762.074,A -85,B 0,C 180,E1 4026.789,E2 4026.789} C_VEL
LIN {X 0,Y 170.724,Z 756.411,A -85,B 0,C 180,E1 4018.978,E2 4018.978} C_VEL
LIN {X 0,Y 178.429,Z 749.493,A -85,B 0,C 180,E1 4012.197,E2 4012.197} C_VEL
LIN {X 0,Y 187.798,Z 740.986,A -85,B 0,C 180,E1 4006.202,E2 4006.202} C_VEL
LIN {X 0,Y 199.128,Z 730.484,A -85,B 0,C 180,E1 4000.696,E2 4000.696} C_VEL
LIN {X 0,Y 210.729,Z 719.194,A -85,B 0,C 180,E1 3996.236,E2 3996.236} C_VEL
LIN {X 0,Y 222.732,Z 706.499,A -85,B 0,C 180,E1 3992.444,E2 3992.444} C_VEL
LIN {X 0,Y 235.598,Z 691.783,A -85,B 0,C 180,E1 3989.047,E2 3989.047} C_VEL
LIN {X 0,Y 247.648,Z 676.54,A -85,B 0,C 180,E1 3986.327,E2 3986.327} C_VEL
LIN {X 0,Y 259.797,Z 659.334,A -85,B 0,C 180,E1 3983.933,E2 3983.933} C_VEL
LIN {X 0,Y 271.139,Z 641.31,A -85,B 0,C 180,E1 3981.965,E2 3981.965} C_VEL
LIN {X 0,Y 281.145,Z 623.018,A -85,B 0,C 180,E1 3980.397,E2 3980.397} C_VEL
LIN {X 0,Y 290.819,Z 602.521,A -85,B 0,C 180,E1 3979.013,E2 3979.013} C_VEL
LIN {X 0,Y 298.98,Z 582.165,A -85,B 0,C 180,E1 3977.935,E2 3977.935} C_VEL
LIN {X 0,Y 305.928,Z 560.633,A -85,B 0,C 180,E1 3977.071,E2 3977.071} C_VEL
LIN {X 0,Y 311.807,Z 537.392,A -85,B 0,C 180,E1 3976.386,E2 3976.386} C_VEL
LIN {X 0,Y 315.91,Z 514.898,A -85,B 0,C 180,E1 3975.89,E2 3975.89} C_VEL
LIN {X 0,Y 325.079,Z 426.987,A -85,B 0,C 180,E1 3974.322,E2 3974.322} C_VEL
LIN {X 0,Y 331.359,Z 365.934,A -85,B 0,C 180,E1 3973.258,E2 3973.258} C_VEL
LIN {X 0,Y 329.353,Z 360.685,A -85,B 0,C 180,E1 3970.495,E2 3970.495} C_VEL
LIN {X 0,Y 328.306,Z 358.031,A -85,B 0,C 180,E1 3968.583,E2 3968.583} C_VEL
LIN {X 0,Y 327.46,Z 355.59,A -85,B 0,C 180,E1 3966.311,E2 3966.311} C_VEL
LIN {X 0,Y 326.994,Z 353.29,A -85,B 0,C 180,E1 3961.752,E2 3961.752} C_VEL
LIN {X 0,Y 327.069,Z 353.344,A -85,B 0,C 180,E1 3960.975,E2 3960.975} C_VEL
LIN {X 0,Y 327.175,Z 354.769,A -85,B 0,C 180,E1 3959.642,E2 3959.642} C_VEL
LIN {X 0,Y 327.332,Z 359.561,A -85,B 0,C 180,E1 3957.657,E2 3957.657} C_VEL
LIN {X 0,Y 327.857,Z 364.476,A -85,B 0,C 180,E1 3955.664,E2 3955.664} C_VEL
LIN {X 0,Y 328.136,Z 365.38,A -85,B 0,C 180,E1 3955.097,E2 3955.097} C_VEL
LIN {X 0,Y 329.818,Z 368.96,A -85,B 0,C 180,E1 3952.598,E2 3952.598} C_VEL
LIN {X 0,Y 330.071,Z 369.755,A -85,B 0,C 180,E1 3952.247,E2 3952.247} C_VEL
LIN {X 0,Y 314.61,Z 512.154,A -85,B 0,C 180,E1 3949.685,E2 3949.685} C_VEL
LIN {X 0,Y 310.433,Z 535.18,A -85,B 0,C 180,E1 3949.183,E2 3949.183} C_VEL
LIN {X 0,Y 305.003,Z 557.065,A -85,B 0,C 180,E1 3948.565,E2 3948.565} C_VEL
LIN {X 0,Y 298.23,Z 578.156,A -85,B 0,C 180,E1 3947.76,E2 3947.76} C_VEL
LIN {X 0,Y 289.736,Z 599.906,A -85,B 0,C 180,E1 3946.689,E2 3946.689} C_VEL
LIN {X 0,Y 280.457,Z 619.997,A -85,B 0,C 180,E1 3945.424,E2 3945.424} C_VEL
LIN {X 0,Y 269.946,Z 639.385,A -85,B 0,C 180,E1 3943.872,E2 3943.872} C_VEL
LIN {X 0,Y 258.386,Z 658.218,A -85,B 0,C 180,E1 3941.967,E2 3941.967} C_VEL
LIN {X 0,Y 246.637,Z 675.118,A -85,B 0,C 180,E1 3939.796,E2 3939.796} C_VEL
LIN {X 0,Y 233.503,Z 692.103,A -85,B 0,C 180,E1 3937.014,E2 3937.014} C_VEL
LIN {X 0,Y 220.612,Z 707.333,A -85,B 0,C 180,E1 3933.812,E2 3933.812} C_VEL
LIN {X 0,Y 207.489,Z 721.421,A -85,B 0,C 180,E1 3929.924,E2 3929.924} C_VEL
LIN {X 0,Y 194.065,Z 734.942,A -85,B 0,C 180,E1 3925.002,E2 3925.002} C_VEL
LIN {X 0,Y 182.478,Z 746.087,A -85,B 0,C 180,E1 3919.606,E2 3919.606} C_VEL
LIN {X 0,Y 172.115,Z 755.766,A -85,B 0,C 180,E1 3913.273,E2 3913.273} C_VEL
LIN {X 0,Y 163.505,Z 764.09,A -85,B 0,C 180,E1 3905.947,E2 3905.947} C_VEL
LIN {X 0,Y 157.58,Z 770.284,A -85,B 0,C 180,E1 3898.416,E2 3898.416} C_VEL
LIN {X 0,Y 153.687,Z 775.289,A -85,B 0,C 180,E1 3889.773,E2 3889.773} C_VEL
LIN {X 0,Y 152.292,Z 778.06,A -85,B 0,C 180,E1 3882.513,E2 3882.513} C_VEL
LIN {X 0,Y 152.017,Z 779.659,A -85,B 0,C 180,E1 3875.283,E2 3875.283} C_VEL
LIN {X 0,Y 152.063,Z 779.959,A -85,B 0,C 180,E1 3869.247,E2 3869.247} C_VEL
LIN {X 0,Y 152.042,Z 779.302,A -85,B 0,C 180,E1 3862.822,E2 3862.822} C_VEL
LIN {X 0,Y 152.47,Z 777.554,A -85,B 0,C 180,E1 3855.958,E2 3855.958} C_VEL
LIN {X 0,Y 154.552,Z 774.03,A -85,B 0,C 180,E1 3847.686,E2 3847.686} C_VEL
LIN {X 0,Y 158.539,Z 769.174,A -85,B 0,C 180,E1 3840.118,E2 3840.118} C_VEL
LIN {X 0,Y 165.612,Z 761.942,A -85,B 0,C 180,E1 3831.99,E2 3831.99} C_VEL
LIN {X 0,Y 174.4,Z 753.596,A -85,B 0,C 180,E1 3825.158,E2 3825.158} C_VEL
LIN {X 0,Y 185.216,Z 743.347,A -85,B 0,C 180,E1 3818.982,E2 3818.982} C_VEL
LIN {X 0,Y 197.186,Z 731.812,A -85,B 0,C 180,E1 3813.741,E2 3813.741} C_VEL
LIN {X 0,Y 209.839,Z 718.842,A -85,B 0,C 180,E1 3809.314,E2 3809.314} C_VEL
LIN {X 0,Y 223.572,Z 703.725,A -85,B 0,C 180,E1 3805.397,E2 3805.397} C_VEL
LIN {X 0,Y 236.633,Z 688.124,A -85,B 0,C 180,E1 3802.282,E2 3802.282} C_VEL
LIN {X 0,Y 249.189,Z 671.35,A -85,B 0,C 180,E1 3799.697,E2 3799.697} C_VEL
LIN {X 0,Y 261.955,Z 652.339,A -85,B 0,C 180,E1 3797.408,E2 3797.408} C_VEL
LIN {X 0,Y 273.069,Z 633.674,A -85,B 0,C 180,E1 3795.643,E2 3795.643} C_VEL
LIN {X 0,Y 283.094,Z 614.127,A -85,B 0,C 180,E1 3794.192,E2 3794.192} C_VEL
LIN {X 0,Y 291.955,Z 594.263,A -85,B 0,C 180,E1 3793.018,E2 3793.018} C_VEL
LIN {X 0,Y 299.323,Z 574.466,A -85,B 0,C 180,E1 3792.098,E2 3792.098} C_VEL
LIN {X 0,Y 306.371,Z 551.246,A -85,B 0,C 180,E1 3791.266,E2 3791.266} C_VEL
LIN {X 0,Y 311.68,Z 528.553,A -85,B 0,C 180,E1 3790.669,E2 3790.669} C_VEL
LIN {X 0,Y 315.285,Z 505.369,A -85,B 0,C 180,E1 3790.193,E2 3790.193} C_VEL
LIN {X 0,Y 329.934,Z 369.394,A -85,B 0,C 180,E1 3787.75,E2 3787.75} C_VEL
LIN {X 0,Y 328.353,Z 366.099,A -85,B 0,C 180,E1 3785.592,E2 3785.592} C_VEL
LIN {X 0,Y 327.207,Z 363.615,A -85,B 0,C 180,E1 3783.504,E2 3783.504} C_VEL
LIN {X 0,Y 325.845,Z 360.838,A -85,B 0,C 180,E1 3778.593,E2 3778.593} C_VEL
LIN {X 0,Y 325.923,Z 362.566,A -85,B 0,C 180,E1 3774.896,E2 3774.896} C_VEL
LIN {X 0,Y 326.536,Z 364.267,A -85,B 0,C 180,E1 3772.699,E2 3772.699} C_VEL
LIN {X 0,Y 327.859,Z 367.919,A -85,B 0,C 180,E1 3769.9,E2 3769.9} C_VEL
LIN {X 0,Y 329.145,Z 371.616,A -85,B 0,C 180,E1 3767.918,E2 3767.918} C_VEL
LIN {X 0,Y 314.004,Z 514.057,A -85,B 0,C 180,E1 3765.449,E2 3765.449} C_VEL
LIN {X 0,Y 309.864,Z 536.745,A -85,B 0,C 180,E1 3764.968,E2 3764.968} C_VEL
LIN {X 0,Y 304.232,Z 559.029,A -85,B 0,C 180,E1 3764.347,E2 3764.347} C_VEL
LIN {X 0,Y 297.598,Z 579.507,A -85,B 0,C 180,E1 3763.574,E2 3763.574} C_VEL
LIN {X 0,Y 289.285,Z 600.438,A -85,B 0,C 180,E1 3762.538,E2 3762.538} C_VEL
LIN {X 0,Y 280.222,Z 619.834,A -85,B 0,C 180,E1 3761.316,E2 3761.316} C_VEL
LIN {X 0,Y 270.059,Z 638.274,A -85,B 0,C 180,E1 3759.836,E2 3759.836} C_VEL
LIN {X 0,Y 257.968,Z 657.508,A -85,B 0,C 180,E1 3757.867,E2 3757.867} C_VEL
LIN {X 0,Y 245.862,Z 674.529,A -85,B 0,C 180,E1 3755.634,E2 3755.634} C_VEL
LIN {X 0,Y 233.249,Z 690.156,A -85,B 0,C 180,E1 3752.974,E2 3752.974} C_VEL
LIN {X 0,Y 220.021,Z 705.042,A -85,B 0,C 180,E1 3749.701,E2 3749.701} C_VEL
LIN {X 0,Y 207.455,Z 717.94,A -85,B 0,C 180,E1 3745.991,E2 3745.991} C_VEL
LIN {X 0,Y 195.211,Z 729.474,A -85,B 0,C 180,E1 3741.594,E2 3741.594} C_VEL
LIN {X 0,Y 183.674,Z 739.791,A -85,B 0,C 180,E1 3736.385,E2 3736.385} C_VEL
LIN {X 0,Y 173.263,Z 748.621,A -85,B 0,C 180,E1 3730.264,E2 3730.264} C_VEL
LIN {X 0,Y 164.509,Z 756.014,A -85,B 0,C 180,E1 3723.161,E2 3723.161} C_VEL
LIN {X 0,Y 158.153,Z 761.704,A -85,B 0,C 180,E1 3715.461,E2 3715.461} C_VEL
LIN {X 0,Y 154.35,Z 765.456,A -85,B 0,C 180,E1 3707.725,E2 3707.725} C_VEL
LIN {X 0,Y 152.505,Z 767.939,A -85,B 0,C 180,E1 3699.433,E2 3699.433} C_VEL
LIN {X 0,Y 152.105,Z 768.771,A -85,B 0,C 180,E1 3693.014,E2 3693.014} C_VEL
LIN {X 0,Y 152.097,Z 768.8,A -85,B 0,C 180,E1 3687.363,E2 3687.363} C_VEL
LIN {X 0,Y 152.45,Z 768.028,A -85,B 0,C 180,E1 3680.944,E2 3680.944} C_VEL
LIN {X 0,Y 154.199,Z 765.668,A -85,B 0,C 180,E1 3672.647,E2 3672.647} C_VEL
LIN {X 0,Y 158.106,Z 761.78,A -85,B 0,C 180,E1 3664.531,E2 3664.531} C_VEL
LIN {X 0,Y 164.439,Z 756.126,A -85,B 0,C 180,E1 3656.823,E2 3656.823} C_VEL
LIN {X 0,Y 173.385,Z 748.591,A -85,B 0,C 180,E1 3649.571,E2 3649.571} C_VEL
LIN {X 0,Y 183.574,Z 739.952,A -85,B 0,C 180,E1 3643.583,E2 3643.583} C_VEL
LIN {X 0,Y 195.356,Z 729.446,A -85,B 0,C 180,E1 3638.265,E2 3638.265} C_VEL
LIN {X 0,Y 208.02,Z 717.501,A -85,B 0,C 180,E1 3633.746,E2 3633.746} C_VEL
LIN {X 0,Y 220.631,Z 704.558,A -85,B 0,C 180,E1 3630.054,E2 3630.054} C_VEL
LIN {X 0,Y 233.278,Z 690.31,A -85,B 0,C 180,E1 3626.939,E2 3626.939} C_VEL
LIN {X 0,Y 246.24,Z 674.234,A -85,B 0,C 180,E1 3624.212,E2 3624.212} C_VEL
LIN {X 0,Y 258.268,Z 657.323,A -85,B 0,C 180,E1 3622.002,E2 3622.002} C_VEL
LIN {X 0,Y 270.334,Z 638.122,A -85,B 0,C 180,E1 3620.046,E2 3620.046} C_VEL
LIN {X 0,Y 280.547,Z 619.565,A -85,B 0,C 180,E1 3618.561,E2 3618.561} C_VEL
LIN {X 0,Y 289.619,Z 600.103,A -85,B 0,C 180,E1 3617.342,E2 3617.342} C_VEL
LIN {X 0,Y 298.26,Z 578.144,A -85,B 0,C 180,E1 3616.269,E2 3616.269} C_VEL
LIN {X 0,Y 305.026,Z 557.057,A -85,B 0,C 180,E1 3615.488,E2 3615.488} C_VEL
LIN {X 0,Y 310.423,Z 535.042,A -85,B 0,C 180,E1 3614.893,E2 3614.893} C_VEL
LIN {X 0,Y 314.511,Z 511.582,A -85,B 0,C 180,E1 3614.408,E2 3614.408} C_VEL
LIN {X 0,Y 329.319,Z 371.589,A -85,B 0,C 180,E1 3611.962,E2 3611.962} C_VEL
LIN {X 0,Y 327.599,Z 366.722,A -85,B 0,C 180,E1 3609.132,E2 3609.132} C_VEL
LIN {X 0,Y 326.441,Z 363.475,A -85,B 0,C 180,E1 3606.154,E2 3606.154} C_VEL
LIN {X 0,Y 326.034,Z 361.219,A -85,B 0,C 180,E1 3601.582,E2 3601.582} C_VEL
LIN {X 0,Y 326.81,Z 362.899,A -85,B 0,C 180,E1 3597.896,E2 3597.896} C_VEL
LIN {X 0,Y 327.855,Z 364.672,A -85,B 0,C 180,E1 3595.628,E2 3595.628} C_VEL
LIN {X 0,Y 328.136,Z 365.38,A -85,B 0,C 180,E1 3595.097,E2 3595.097} C_VEL
LIN {X 0,Y 328.348,Z 367.054,A -85,B 0,C 180,E1 3594.537,E2 3594.537} C_VEL
LIN {X 0,Y 328.294,Z 371.151,A -85,B 0,C 180,E1 3593.969,E2 3593.969} C_VEL
LIN {X 0,Y 327.868,Z 377.152,A -85,B 0,C 180,E1 3593.589,E2 3593.589} C_VEL
LIN {X 0,Y 326.859,Z 387.092,A -85,B 0,C 180,E1 3593.322,E2 3593.322} C_VEL
LIN {X 0,Y 312.924,Z 512.587,A -85,B 0,C 180,E1 3591.111,E2 3591.111} C_VEL
LIN {X 0,Y 308.692,Z 535.407,A -85,B 0,C 180,E1 3590.63,E2 3590.63} C_VEL
LIN {X 0,Y 303.033,Z 557.71,A -85,B 0,C 180,E1 3590.022,E2 3590.022} C_VEL
LIN {X 0,Y 296.151,Z 578.72,A -85,B 0,C 180,E1 3589.246,E2 3589.246} C_VEL
LIN {X 0,Y 287.511,Z 600.341,A -85,B 0,C 180,E1 3588.217,E2 3588.217} C_VEL
LIN {X 0,Y 278.081,Z 620.337,A -85,B 0,C 180,E1 3587,E2 3587} C_VEL
LIN {X 0,Y 267.455,Z 639.478,A -85,B 0,C 180,E1 3585.517,E2 3585.517} C_VEL
LIN {X 0,Y 255.745,Z 658.109,A -85,B 0,C 180,E1 3583.694,E2 3583.694} C_VEL
LIN {X 0,Y 243.654,Z 675.061,A -85,B 0,C 180,E1 3581.581,E2 3581.581} C_VEL
LIN {X 0,Y 230.102,Z 692.08,A -85,B 0,C 180,E1 3578.86,E2 3578.86} C_VEL
LIN {X 0,Y 217.055,Z 706.988,A -85,B 0,C 180,E1 3575.791,E2 3575.791} C_VEL
LIN {X 0,Y 203.714,Z 720.792,A -85,B 0,C 180,E1 3572.06,E2 3572.06} C_VEL
LIN {X 0,Y 190.023,Z 734.035,A -85,B 0,C 180,E1 3567.337,E2 3567.337} C_VEL
LIN {X 0,Y 177.72,Z 745.24,A -85,B 0,C 180,E1 3561.964,E2 3561.964} C_VEL
LIN {X 0,Y 166.585,Z 755.036,A -85,B 0,C 180,E1 3555.58,E2 3555.58} C_VEL
LIN {X 0,Y 157.559,Z 763.149,A -85,B 0,C 180,E1 3548.454,E2 3548.454} C_VEL
LIN {X 0,Y 150.584,Z 769.713,A -85,B 0,C 180,E1 3540.306,E2 3540.306} C_VEL
LIN {X 0,Y 146.104,Z 774.82,A -85,B 0,C 180,E1 3531.266,E2 3531.266} C_VEL
LIN {X 0,Y 144.407,Z 777.642,A -85,B 0,C 180,E1 3523.616,E2 3523.616} C_VEL
LIN {X 0,Y 144.024,Z 779.312,A -85,B 0,C 180,E1 3515.977,E2 3515.977} C_VEL
LIN {X 0,Y 144.071,Z 779.692,A -85,B 0,C 180,E1 3509.602,E2 3509.602} C_VEL
LIN {X 0,Y 144.045,Z 779.082,A -85,B 0,C 180,E1 3502.823,E2 3502.823} C_VEL
LIN {X 0,Y 144.504,Z 777.393,A -85,B 0,C 180,E1 3495.623,E2 3495.623} C_VEL
LIN {X 0,Y 146.678,Z 774.096,A -85,B 0,C 180,E1 3487.136,E2 3487.136} C_VEL
LIN {X 0,Y 151.377,Z 768.87,A -85,B 0,C 180,E1 3478.548,E2 3478.548} C_VEL
LIN {X 0,Y 159.098,Z 761.632,A -85,B 0,C 180,E1 3470.133,E2 3470.133} C_VEL
LIN {X 0,Y 168.549,Z 753.286,A -85,B 0,C 180,E1 3463.144,E2 3463.144} C_VEL
LIN {X 0,Y 180.052,Z 743.03,A -85,B 0,C 180,E1 3456.905,E2 3456.905} C_VEL
LIN {X 0,Y 192.906,Z 731.229,A -85,B 0,C 180,E1 3451.567,E2 3451.567} C_VEL
LIN {X 0,Y 205.869,Z 718.511,A -85,B 0,C 180,E1 3447.282,E2 3447.282} C_VEL
LIN {X 0,Y 219.347,Z 704.241,A -85,B 0,C 180,E1 3443.623,E2 3443.623} C_VEL
LIN {X 0,Y 232.793,Z 688.745,A -85,B 0,C 180,E1 3440.562,E2 3440.562} C_VEL
LIN {X 0,Y 245.83,Z 671.886,A -85,B 0,C 180,E1 3438.005,E2 3438.005} C_VEL
LIN {X 0,Y 258.74,Z 653.264,A -85,B 0,C 180,E1 3435.806,E2 3435.806} C_VEL
LIN {X 0,Y 269.521,Z 635.655,A -85,B 0,C 180,E1 3434.172,E2 3434.172} C_VEL
LIN {X 0,Y 280.282,Z 615.448,A -85,B 0,C 180,E1 3432.692,E2 3432.692} C_VEL
LIN {X 0,Y 289.509,Z 595.402,A -85,B 0,C 180,E1 3431.534,E2 3431.534} C_VEL
LIN {X 0,Y 297.346,Z 574.782,A -85,B 0,C 180,E1 3430.607,E2 3430.607} C_VEL
LIN {X 0,Y 304.523,Z 551.607,A -85,B 0,C 180,E1 3429.806,E2 3429.806} C_VEL
LIN {X 0,Y 309.893,Z 529.075,A -85,B 0,C 180,E1 3429.235,E2 3429.235} C_VEL
LIN {X 0,Y 313.587,Z 505.955,A -85,B 0,C 180,E1 3428.772,E2 3428.772} C_VEL
LIN {X 0,Y 327.943,Z 375.424,A -85,B 0,C 180,E1 3426.477,E2 3426.477} C_VEL
LIN {X 0,Y 326.132,Z 371.488,A -85,B 0,C 180,E1 3423.339,E2 3423.339} C_VEL
LIN {X 0,Y 324.87,Z 368.782,A -85,B 0,C 180,E1 3418.589,E2 3418.589} C_VEL
LIN {X 0,Y 325.018,Z 370.776,A -85,B 0,C 180,E1 3414.527,E2 3414.527} C_VEL
LIN {X 0,Y 325.524,Z 372.3,A -85,B 0,C 180,E1 3412.765,E2 3412.765} C_VEL
LIN {X 0,Y 326.669,Z 375.608,A -85,B 0,C 180,E1 3410.228,E2 3410.228} C_VEL
LIN {X 0,Y 327.257,Z 377.415,A -85,B 0,C 180,E1 3409.205,E2 3409.205} C_VEL
LIN {X 0,Y 312.388,Z 514.012,A -85,B 0,C 180,E1 3406.887,E2 3406.887} C_VEL
LIN {X 0,Y 308.185,Z 536.668,A -85,B 0,C 180,E1 3406.424,E2 3406.424} C_VEL
LIN {X 0,Y 302.423,Z 559.103,A -85,B 0,C 180,E1 3405.825,E2 3405.825} C_VEL
LIN {X 0,Y 295.444,Z 580.242,A -85,B 0,C 180,E1 3405.056,E2 3405.056} C_VEL
LIN {X 0,Y 286.988,Z 601.019,A -85,B 0,C 180,E1 3404.06,E2 3404.06} C_VEL
LIN {X 0,Y 277.758,Z 620.318,A -85,B 0,C 180,E1 3402.883,E2 3402.883} C_VEL
LIN {X 0,Y 267.598,Z 638.378,A -85,B 0,C 180,E1 3401.482,E2 3401.482} C_VEL
LIN {X 0,Y 255.451,Z 657.313,A -85,B 0,C 180,E1 3399.613,E2 3399.613} C_VEL
LIN {X 0,Y 243.042,Z 674.362,A -85,B 0,C 180,E1 3397.451,E2 3397.451} C_VEL
LIN {X 0,Y 229.819,Z 690.338,A -85,B 0,C 180,E1 3394.811,E2 3394.811} C_VEL
LIN {X 0,Y 215.67,Z 705.728,A -85,B 0,C 180,E1 3391.476,E2 3391.476} C_VEL
LIN {X 0,Y 202.305,Z 718.949,A -85,B 0,C 180,E1 3387.684,E2 3387.684} C_VEL
LIN {X 0,Y 189.596,Z 730.344,A -85,B 0,C 180,E1 3383.28,E2 3383.28} C_VEL
LIN {X 0,Y 176.987,Z 740.984,A -85,B 0,C 180,E1 3377.735,E2 3377.735} C_VEL
LIN {X 0,Y 166.146,Z 749.709,A -85,B 0,C 180,E1 3371.449,E2 3371.449} C_VEL
LIN {X 0,Y 157.03,Z 756.858,A -85,B 0,C 180,E1 3364.131,E2 3364.131} C_VEL
LIN {X 0,Y 150.323,Z 762.393,A -85,B 0,C 180,E1 3356.039,E2 3356.039} C_VEL
LIN {X 0,Y 146.359,Z 766.055,A -85,B 0,C 180,E1 3347.903,E2 3347.903} C_VEL
LIN {X 0,Y 144.473,Z 768.357,A -85,B 0,C 180,E1 3339.159,E2 3339.159} C_VEL
LIN {X 0,Y 144.099,Z 769.104,A -85,B 0,C 180,E1 3332.386,E2 3332.386} C_VEL
LIN {X 0,Y 144.134,Z 769.03,A -85,B 0,C 180,E1 3326.022,E2 3326.022} C_VEL
LIN {X 0,Y 144.78,Z 767.961,A -85,B 0,C 180,E1 3318.447,E2 3318.447} C_VEL
LIN {X 0,Y 147.065,Z 765.359,A -85,B 0,C 180,E1 3310.127,E2 3310.127} C_VEL
LIN {X 0,Y 152.106,Z 760.911,A -85,B 0,C 180,E1 3301.325,E2 3301.325} C_VEL
LIN {X 0,Y 159.571,Z 754.968,A -85,B 0,C 180,E1 3293.47,E2 3293.47} C_VEL
LIN {X 0,Y 168.954,Z 747.505,A -85,B 0,C 180,E1 3286.649,E2 3286.649} C_VEL
LIN {X 0,Y 180.325,Z 738.341,A -85,B 0,C 180,E1 3280.57,E2 3280.57} C_VEL
LIN {X 0,Y 192.327,Z 728.09,A -85,B 0,C 180,E1 3275.61,E2 3275.61} C_VEL
LIN {X 0,Y 205.712,Z 715.765,A -85,B 0,C 180,E1 3271.194,E2 3271.194} C_VEL
LIN {X 0,Y 218.921,Z 702.576,A -85,B 0,C 180,E1 3267.623,E2 3267.623} C_VEL
LIN {X 0,Y 232.079,Z 687.92,A -85,B 0,C 180,E1 3264.63,E2 3264.63} C_VEL
LIN {X 0,Y 245.801,Z 670.907,A -85,B 0,C 180,E1 3261.963,E2 3261.963} C_VEL
LIN {X 0,Y 257.849,Z 654.165,A -85,B 0,C 180,E1 3259.928,E2 3259.928} C_VEL
LIN {X 0,Y 268.977,Z 636.383,A -85,B 0,C 180,E1 3258.244,E2 3258.244} C_VEL
LIN {X 0,Y 279.848,Z 616.532,A -85,B 0,C 180,E1 3256.764,E2 3256.764} C_VEL
LIN {X 0,Y 288.671,Z 597.684,A -85,B 0,C 180,E1 3255.663,E2 3255.663} C_VEL
LIN {X 0,Y 296.696,Z 577.244,A -85,B 0,C 180,E1 3254.726,E2 3254.726} C_VEL
LIN {X 0,Y 303.453,Z 556.417,A -85,B 0,C 180,E1 3253.992,E2 3253.992} C_VEL
LIN {X 0,Y 308.887,Z 534.377,A -85,B 0,C 180,E1 3253.427,E2 3253.427} C_VEL
LIN {X 0,Y 313.097,Z 510.057,A -85,B 0,C 180,E1 3252.945,E2 3252.945} C_VEL
LIN {X 0,Y 327.456,Z 377.451,A -85,B 0,C 180,E1 3250.69,E2 3250.69} C_VEL
LIN {X 0,Y 326.195,Z 373.846,A -85,B 0,C 180,E1 3248.283,E2 3248.283} C_VEL
LIN {X 0,Y 325.376,Z 371.25,A -85,B 0,C 180,E1 3245.82,E2 3245.82} C_VEL
LIN {X 0,Y 325.063,Z 369.158,A -85,B 0,C 180,E1 3241.546,E2 3241.546} C_VEL
LIN {X 0,Y 325.966,Z 371.101,A -85,B 0,C 180,E1 3237.539,E2 3237.539} C_VEL
LIN {X 0,Y 326.762,Z 372.586,A -85,B 0,C 180,E1 3235.789,E2 3235.789} C_VEL
LIN {X 0,Y 328.111,Z 375.695,A -85,B 0,C 180,E1 3233.521,E2 3233.521} C_VEL
LIN {X 0,Y 326.859,Z 387.092,A -85,B 0,C 180,E1 3233.322,E2 3233.322} C_VEL
LIN {X 0,Y 325.86,Z 394.791,A -85,B 0,C 180,E1 3233.361,E2 3233.361} C_VEL
LIN {X 0,Y 322.649,Z 415.373,A -85,B 0,C 180,E1 3234.107,E2 3234.107} C_VEL
LIN {X 0,Y 321.802,Z 421.977,A -85,B 0,C 180,E1 3234.126,E2 3234.126} C_VEL
LIN {X 0,Y 311.391,Z 513.344,A -85,B 0,C 180,E1 3232.546,E2 3232.546} C_VEL
LIN {X 0,Y 307.034,Z 536.171,A -85,B 0,C 180,E1 3232.079,E2 3232.079} C_VEL
LIN {X 0,Y 301.088,Z 558.906,A -85,B 0,C 180,E1 3231.479,E2 3231.479} C_VEL
LIN {X 0,Y 294.275,Z 579.285,A -85,B 0,C 180,E1 3230.753,E2 3230.753} C_VEL
LIN {X 0,Y 285.493,Z 600.777,A -85,B 0,C 180,E1 3229.767,E2 3229.767} C_VEL
LIN {X 0,Y 275.775,Z 620.946,A -85,B 0,C 180,E1 3228.584,E2 3228.584} C_VEL
LIN {X 0,Y 265.025,Z 639.848,A -85,B 0,C 180,E1 3227.168,E2 3227.168} C_VEL
LIN {X 0,Y 252.448,Z 659.262,A -85,B 0,C 180,E1 3225.317,E2 3225.317} C_VEL
LIN {X 0,Y 240.128,Z 676.047,A -85,B 0,C 180,E1 3223.268,E2 3223.268} C_VEL
LIN {X 0,Y 226.482,Z 692.586,A -85,B 0,C 180,E1 3220.665,E2 3220.665} C_VEL
LIN {X 0,Y 212.976,Z 707.485,A -85,B 0,C 180,E1 3217.642,E2 3217.642} C_VEL
LIN {X 0,Y 199.183,Z 721.183,A -85,B 0,C 180,E1 3213.964,E2 3213.964} C_VEL
LIN {X 0,Y 184.263,Z 734.9,A -85,B 0,C 180,E1 3209.017,E2 3209.017} C_VEL
LIN {X 0,Y 171.122,Z 746.274,A -85,B 0,C 180,E1 3203.418,E2 3203.418} C_VEL
LIN {X 0,Y 159.293,Z 755.991,A -85,B 0,C 180,E1 3196.727,E2 3196.727} C_VEL
LIN {X 0,Y 149.117,Z 764.436,A -85,B 0,C 180,E1 3188.577,E2 3188.577} C_VEL
LIN {X 0,Y 142.109,Z 770.746,A -85,B 0,C 180,E1 3179.969,E2 3179.969} C_VEL
LIN {X 0,Y 138.023,Z 775.033,A -85,B 0,C 180,E1 3171.235,E2 3171.235} C_VEL
LIN {X 0,Y 136.294,Z 777.849,A -85,B 0,C 180,E1 3162.662,E2 3162.662} C_VEL
LIN {X 0,Y 136.026,Z 779.13,A -85,B 0,C 180,E1 3155.06,E2 3155.06} C_VEL
LIN {X 0,Y 136.069,Z 779.353,A -85,B 0,C 180,E1 3148.737,E2 3148.737} C_VEL
LIN {X 0,Y 136.055,Z 778.715,A -85,B 0,C 180,E1 3141.974,E2 3141.974} C_VEL
LIN {X 0,Y 136.62,Z 777.083,A -85,B 0,C 180,E1 3134.725,E2 3134.725} C_VEL
LIN {X 0,Y 139.11,Z 773.794,A -85,B 0,C 180,E1 3125.815,E2 3125.815} C_VEL
LIN {X 0,Y 144.334,Z 768.565,A -85,B 0,C 180,E1 3116.822,E2 3116.822} C_VEL
LIN {X 0,Y 152.762,Z 761.323,A -85,B 0,C 180,E1 3108.118,E2 3108.118} C_VEL
LIN {X 0,Y 162.919,Z 752.975,A -85,B 0,C 180,E1 3100.988,E2 3100.988} C_VEL
LIN {X 0,Y 175.137,Z 742.713,A -85,B 0,C 180,E1 3094.707,E2 3094.707} C_VEL
LIN {X 0,Y 188.376,Z 731.156,A -85,B 0,C 180,E1 3089.489,E2 3089.489} C_VEL
LIN {X 0,Y 201.416,Z 718.898,A -85,B 0,C 180,E1 3085.385,E2 3085.385} C_VEL
LIN {X 0,Y 216.135,Z 703.891,A -85,B 0,C 180,E1 3081.594,E2 3081.594} C_VEL
LIN {X 0,Y 230,Z 688.386,A -85,B 0,C 180,E1 3078.619,E2 3078.619} C_VEL
LIN {X 0,Y 243.066,Z 671.929,A -85,B 0,C 180,E1 3076.204,E2 3076.204} C_VEL
LIN {X 0,Y 256.172,Z 653.51,A -85,B 0,C 180,E1 3074.097,E2 3074.097} C_VEL
LIN {X 0,Y 267.299,Z 635.736,A -85,B 0,C 180,E1 3072.507,E2 3072.507} C_VEL
LIN {X 0,Y 278.157,Z 615.783,A -85,B 0,C 180,E1 3071.1,E2 3071.1} C_VEL
LIN {X 0,Y 287.33,Z 596.291,A -85,B 0,C 180,E1 3070.015,E2 3070.015} C_VEL
LIN {X 0,Y 295.405,Z 575.563,A -85,B 0,C 180,E1 3069.114,E2 3069.114} C_VEL
LIN {X 0,Y 302.572,Z 553.097,A -85,B 0,C 180,E1 3068.36,E2 3068.36} C_VEL
LIN {X 0,Y 307.919,Z 531.288,A -85,B 0,C 180,E1 3067.821,E2 3067.821} C_VEL
LIN {X 0,Y 311.882,Z 508.066,A -85,B 0,C 180,E1 3067.365,E2 3067.365} C_VEL
LIN {X 0,Y 326.074,Z 381.798,A -85,B 0,C 180,E1 3065.19,E2 3065.19} C_VEL
LIN {X 0,Y 324.978,Z 379.245,A -85,B 0,C 180,E1 3062.998,E2 3062.998} C_VEL
LIN {X 0,Y 323.895,Z 376.726,A -85,B 0,C 180,E1 3058.585,E2 3058.585} C_VEL
LIN {X 0,Y 324.089,Z 378.89,A -85,B 0,C 180,E1 3054.334,E2 3054.334} C_VEL
LIN {X 0,Y 324.573,Z 380.54,A -85,B 0,C 180,E1 3052.655,E2 3052.655} C_VEL
LIN {X 0,Y 325.516,Z 383.385,A -85,B 0,C 180,E1 3050.504,E2 3050.504} C_VEL
LIN {X 0,Y 310.976,Z 513.929,A -85,B 0,C 180,E1 3048.339,E2 3048.339} C_VEL
LIN {X 0,Y 306.706,Z 536.59,A -85,B 0,C 180,E1 3047.895,E2 3047.895} C_VEL
LIN {X 0,Y 300.973,Z 558.68,A -85,B 0,C 180,E1 3047.334,E2 3047.334} C_VEL
LIN {X 0,Y 293.944,Z 579.703,A -85,B 0,C 180,E1 3046.608,E2 3046.608} C_VEL
LIN {X 0,Y 285.348,Z 600.605,A -85,B 0,C 180,E1 3045.656,E2 3045.656} C_VEL
LIN {X 0,Y 275.952,Z 619.997,A -85,B 0,C 180,E1 3044.53,E2 3044.53} C_VEL
LIN {X 0,Y 265.035,Z 639.026,A -85,B 0,C 180,E1 3043.113,E2 3043.113} C_VEL
LIN {X 0,Y 252.333,Z 658.296,A -85,B 0,C 180,E1 3041.262,E2 3041.262} C_VEL
LIN {X 0,Y 239.638,Z 675.267,A -85,B 0,C 180,E1 3039.161,E2 3039.161} C_VEL
LIN {X 0,Y 226.483,Z 690.683,A -85,B 0,C 180,E1 3036.669,E2 3036.669} C_VEL
LIN {X 0,Y 212.266,Z 705.698,A -85,B 0,C 180,E1 3033.502,E2 3033.502} C_VEL
LIN {X 0,Y 198.784,Z 718.587,A -85,B 0,C 180,E1 3029.895,E2 3029.895} C_VEL
LIN {X 0,Y 185.283,Z 730.266,A -85,B 0,C 180,E1 3025.485,E2 3025.485} C_VEL
LIN {X 0,Y 172.177,Z 740.843,A -85,B 0,C 180,E1 3020.043,E2 3020.043} C_VEL
LIN {X 0,Y 160.594,Z 749.621,A -85,B 0,C 180,E1 3013.715,E2 3013.715} C_VEL
LIN {X 0,Y 150.667,Z 756.903,A -85,B 0,C 180,E1 3006.2,E2 3006.2} C_VEL
LIN {X 0,Y 143.308,Z 762.493,A -85,B 0,C 180,E1 2997.869,E2 2997.869} C_VEL
LIN {X 0,Y 138.802,Z 766.208,A -85,B 0,C 180,E1 2989.324,E2 2989.324} C_VEL
LIN {X 0,Y 136.587,Z 768.587,A -85,B 0,C 180,E1 2980.118,E2 2980.118} C_VEL
LIN {X 0,Y 136.113,Z 769.374,A -85,B 0,C 180,E1 2972.947,E2 2972.947} C_VEL
LIN {X 0,Y 136.121,Z 769.361,A -85,B 0,C 180,E1 2966.631,E2 2966.631} C_VEL
LIN {X 0,Y 136.688,Z 768.487,A -85,B 0,C 180,E1 2959.037,E2 2959.037} C_VEL
LIN {X 0,Y 139.103,Z 765.956,A -85,B 0,C 180,E1 2949.818,E2 2949.818} C_VEL
LIN {X 0,Y 144.098,Z 761.938,A -85,B 0,C 180,E1 2940.942,E2 2940.942} C_VEL
LIN {X 0,Y 151.806,Z 756.138,A -85,B 0,C 180,E1 2932.704,E2 2932.704} C_VEL
LIN {X 0,Y 162.427,Z 748.299,A -85,B 0,C 180,E1 2925.066,E2 2925.066} C_VEL
LIN {X 0,Y 173.888,Z 739.646,A -85,B 0,C 180,E1 2919.084,E2 2919.084} C_VEL
LIN {X 0,Y 186.736,Z 729.172,A -85,B 0,C 180,E1 2913.911,E2 2913.911} C_VEL
LIN {X 0,Y 200.869,Z 716.767,A -85,B 0,C 180,E1 2909.417,E2 2909.417} C_VEL
LIN {X 0,Y 214.488,Z 703.69,A -85,B 0,C 180,E1 2905.886,E2 2905.886} C_VEL
LIN {X 0,Y 228.002,Z 689.173,A -85,B 0,C 180,E1 2902.944,E2 2902.944} C_VEL
LIN {X 0,Y 241.632,Z 672.917,A -85,B 0,C 180,E1 2900.411,E2 2900.411} C_VEL
LIN {X 0,Y 253.96,Z 656.298,A -85,B 0,C 180,E1 2898.413,E2 2898.413} C_VEL
LIN {X 0,Y 265.487,Z 638.614,A -85,B 0,C 180,E1 2896.75,E2 2896.75} C_VEL
LIN {X 0,Y 276.308,Z 619.706,A -85,B 0,C 180,E1 2895.348,E2 2895.348} C_VEL
LIN {X 0,Y 285.713,Z 600.244,A -85,B 0,C 180,E1 2894.225,E2 2894.225} C_VEL
LIN {X 0,Y 294.408,Z 578.982,A -85,B 0,C 180,E1 2893.266,E2 2893.266} C_VEL
LIN {X 0,Y 301.398,Z 557.989,A -85,B 0,C 180,E1 2892.547,E2 2892.547} C_VEL
LIN {X 0,Y 307.088,Z 535.815,A -85,B 0,C 180,E1 2891.992,E2 2891.992} C_VEL
LIN {X 0,Y 311.312,Z 512.977,A -85,B 0,C 180,E1 2891.548,E2 2891.548} C_VEL
LIN {X 0,Y 325.724,Z 383.575,A -85,B 0,C 180,E1 2889.405,E2 2889.405} C_VEL
LIN {X 0,Y 324.693,Z 380.323,A -85,B 0,C 180,E1 2886.898,E2 2886.898} C_VEL
LIN {X 0,Y 324.279,Z 378.915,A -85,B 0,C 180,E1 2885.308,E2 2885.308} C_VEL
LIN {X 0,Y 324.101,Z 377.095,A -85,B 0,C 180,E1 2881.414,E2 2881.414} C_VEL
LIN {X 0,Y 325.44,Z 379.805,A -85,B 0,C 180,E1 2876.477,E2 2876.477} C_VEL
LIN {X 0,Y 326.259,Z 382.147,A -85,B 0,C 180,E1 2874.801,E2 2874.801} C_VEL
LIN {X 0,Y 321.802,Z 421.977,A -85,B 0,C 180,E1 2874.126,E2 2874.126} C_VEL
LIN {X 0,Y 320.8,Z 429.672,A -85,B 0,C 180,E1 2874.169,E2 2874.169} C_VEL
LIN {X 0,Y 317.65,Z 450.246,A -85,B 0,C 180,E1 2874.938,E2 2874.938} C_VEL
LIN {X 0,Y 316.804,Z 456.852,A -85,B 0,C 180,E1 2874.966,E2 2874.966} C_VEL
LIN {X 0,Y 309.967,Z 514.706,A -85,B 0,C 180,E1 2873.983,E2 2873.983} C_VEL
LIN {X 0,Y 305.425,Z 537.593,A -85,B 0,C 180,E1 2873.529,E2 2873.529} C_VEL
LIN {X 0,Y 299.217,Z 560.495,A -85,B 0,C 180,E1 2872.942,E2 2872.942} C_VEL
LIN {X 0,Y 292.133,Z 581.15,A -85,B 0,C 180,E1 2872.23,E2 2872.23} C_VEL
LIN {X 0,Y 283.22,Z 602.23,A -85,B 0,C 180,E1 2871.289,E2 2871.289} C_VEL
LIN {X 0,Y 273.468,Z 621.894,A -85,B 0,C 180,E1 2870.171,E2 2870.171} C_VEL
LIN {X 0,Y 262.909,Z 640.069,A -85,B 0,C 180,E1 2868.861,E2 2868.861} C_VEL
LIN {X 0,Y 249.813,Z 659.787,A -85,B 0,C 180,E1 2867.048,E2 2867.048} C_VEL
LIN {X 0,Y 236.999,Z 676.796,A -85,B 0,C 180,E1 2865.035,E2 2865.035} C_VEL
LIN {X 0,Y 223.093,Z 693.093,A -85,B 0,C 180,E1 2862.526,E2 2862.526} C_VEL
LIN {X 0,Y 209.127,Z 707.943,A -85,B 0,C 180,E1 2859.565,E2 2859.565} C_VEL
LIN {X 0,Y 194.881,Z 721.574,A -85,B 0,C 180,E1 2855.954,E2 2855.954} C_VEL
LIN {X 0,Y 180.082,Z 734.583,A -85,B 0,C 180,E1 2851.31,E2 2851.31} C_VEL
LIN {X 0,Y 166.612,Z 745.673,A -85,B 0,C 180,E1 2845.907,E2 2845.907} C_VEL
LIN {X 0,Y 154.201,Z 755.262,A -85,B 0,C 180,E1 2839.343,E2 2839.343} C_VEL
LIN {X 0,Y 143.513,Z 763.496,A -85,B 0,C 180,E1 2831.441,E2 2831.441} C_VEL
LIN {X 0,Y 135.815,Z 769.68,A -85,B 0,C 180,E1 2822.939,E2 2822.939} C_VEL
LIN {X 0,Y 130.54,Z 774.564,A -85,B 0,C 180,E1 2812.993,E2 2812.993} C_VEL
LIN {X 0,Y 128.486,Z 777.295,A -85,B 0,C 180,E1 2804.419,E2 2804.419} C_VEL
LIN {X 0,Y 128.031,Z 778.811,A -85,B 0,C 180,E1 2795.827,E2 2795.827} C_VEL
LIN {X 0,Y 128.076,Z 779.087,A -85,B 0,C 180,E1 2789.105,E2 2789.105} C_VEL
LIN {X 0,Y 128.058,Z 778.495,A -85,B 0,C 180,E1 2781.921,E2 2781.921} C_VEL
LIN {X 0,Y 128.682,Z 776.908,A -85,B 0,C 180,E1 2774.22,E2 2774.22} C_VEL
LIN {X 0,Y 131.362,Z 773.737,A -85,B 0,C 180,E1 2764.925,E2 2764.925} C_VEL
LIN {X 0,Y 136.864,Z 768.728,A -85,B 0,C 180,E1 2755.64,E2 2755.64} C_VEL
LIN {X 0,Y 145.261,Z 762.12,A -85,B 0,C 180,E1 2747.046,E2 2747.046} C_VEL
LIN {X 0,Y 155.843,Z 753.927,A -85,B 0,C 180,E1 2739.657,E2 2739.657} C_VEL
LIN {X 0,Y 169.219,Z 743.429,A -85,B 0,C 180,E1 2732.928,E2 2732.928} C_VEL
LIN {X 0,Y 183.056,Z 732.021,A -85,B 0,C 180,E1 2727.663,E2 2727.663} C_VEL
LIN {X 0,Y 197.193,Z 719.286,A -85,B 0,C 180,E1 2723.404,E2 2723.404} C_VEL
LIN {X 0,Y 212.381,Z 704.407,A -85,B 0,C 180,E1 2719.688,E2 2719.688} C_VEL
LIN {X 0,Y 226.197,Z 689.446,A -85,B 0,C 180,E1 2716.87,E2 2716.87} C_VEL
LIN {X 0,Y 239.782,Z 672.957,A -85,B 0,C 180,E1 2714.488,E2 2714.488} C_VEL
LIN {X 0,Y 252.941,Z 655.113,A -85,B 0,C 180,E1 2712.487,E2 2712.487} C_VEL
LIN {X 0,Y 264.785,Z 636.667,A -85,B 0,C 180,E1 2710.883,E2 2710.883} C_VEL
LIN {X 0,Y 276.119,Z 616.379,A -85,B 0,C 180,E1 2709.501,E2 2709.501} C_VEL
LIN {X 0,Y 285.493,Z 596.844,A -85,B 0,C 180,E1 2708.458,E2 2708.458} C_VEL
LIN {X 0,Y 293.539,Z 576.694,A -85,B 0,C 180,E1 2707.615,E2 2707.615} C_VEL
LIN {X 0,Y 300.754,Z 554.819,A -85,B 0,C 180,E1 2706.902,E2 2706.902} C_VEL
LIN {X 0,Y 306.311,Z 532.727,A -85,B 0,C 180,E1 2706.374,E2 2706.374} C_VEL
LIN {X 0,Y 310.556,Z 508.777,A -85,B 0,C 180,E1 2705.918,E2 2705.918} C_VEL
LIN {X 0,Y 324.374,Z 388.225,A -85,B 0,C 180,E1 2703.888,E2 2703.888} C_VEL
LIN {X 0,Y 323.629,Z 386.658,A -85,B 0,C 180,E1 2702.124,E2 2702.124} C_VEL
LIN {X 0,Y 322.903,Z 384.671,A -85,B 0,C 180,E1 2698.403,E2 2698.403} C_VEL
LIN {X 0,Y 323.304,Z 387.484,A -85,B 0,C 180,E1 2693.607,E2 2693.607} C_VEL
LIN {X 0,Y 323.895,Z 389.809,A -85,B 0,C 180,E1 2691.807,E2 2691.807} C_VEL
LIN {X 0,Y 309.755,Z 513.921,A -85,B 0,C 180,E1 2689.803,E2 2689.803} C_VEL
LIN {X 0,Y 305.432,Z 536.511,A -85,B 0,C 180,E1 2689.378,E2 2689.378} C_VEL
LIN {X 0,Y 299.489,Z 559.028,A -85,B 0,C 180,E1 2688.835,E2 2688.835} C_VEL
LIN {X 0,Y 292.623,Z 579.277,A -85,B 0,C 180,E1 2688.169,E2 2688.169} C_VEL
LIN {X 0,Y 283.932,Z 600.19,A -85,B 0,C 180,E1 2687.27,E2 2687.27} C_VEL
LIN {X 0,Y 274.377,Z 619.661,A -85,B 0,C 180,E1 2686.198,E2 2686.198} C_VEL
LIN {X 0,Y 263.573,Z 638.24,A -85,B 0,C 180,E1 2684.887,E2 2684.887} C_VEL
LIN {X 0,Y 251.178,Z 656.89,A -85,B 0,C 180,E1 2683.201,E2 2683.201} C_VEL
LIN {X 0,Y 238.593,Z 673.476,A -85,B 0,C 180,E1 2681.273,E2 2681.273} C_VEL
LIN {X 0,Y 225.057,Z 689.208,A -85,B 0,C 180,E1 2678.898,E2 2678.898} C_VEL
LIN {X 0,Y 211.158,Z 703.756,A -85,B 0,C 180,E1 2676.043,E2 2676.043} C_VEL
LIN {X 0,Y 197.083,Z 716.849,A -85,B 0,C 180,E1 2672.598,E2 2672.598} C_VEL
LIN {X 0,Y 182.395,Z 729.288,A -85,B 0,C 180,E1 2668.175,E2 2668.175} C_VEL
LIN {X 0,Y 168.934,Z 739.783,A -85,B 0,C 180,E1 2663.034,E2 2663.034} C_VEL
LIN {X 0,Y 156.404,Z 748.747,A -85,B 0,C 180,E1 2656.782,E2 2656.782} C_VEL
LIN {X 0,Y 144.863,Z 756.713,A -85,B 0,C 180,E1 2648.744,E2 2648.744} C_VEL
LIN {X 0,Y 136.754,Z 762.386,A -85,B 0,C 180,E1 2640.296,E2 2640.296} C_VEL
LIN {X 0,Y 131.35,Z 766.344,A -85,B 0,C 180,E1 2630.963,E2 2630.963} C_VEL
LIN {X 0,Y 128.73,Z 768.817,A -85,B 0,C 180,E1 2621.196,E2 2621.196} C_VEL
LIN {X 0,Y 128.133,Z 769.644,A -85,B 0,C 180,E1 2613.579,E2 2613.579} C_VEL
LIN {X 0,Y 128.114,Z 769.694,A -85,B 0,C 180,E1 2607.316,E2 2607.316} C_VEL
LIN {X 0,Y 128.538,Z 769.03,A -85,B 0,C 180,E1 2600.147,E2 2600.147} C_VEL
LIN {X 0,Y 130.654,Z 767.006,A -85,B 0,C 180,E1 2590.788,E2 2590.788} C_VEL
LIN {X 0,Y 135.398,Z 763.328,A -85,B 0,C 180,E1 2581.495,E2 2581.495} C_VEL
LIN {X 0,Y 143.647,Z 757.601,A -85,B 0,C 180,E1 2572.229,E2 2572.229} C_VEL
LIN {X 0,Y 154.158,Z 750.459,A -85,B 0,C 180,E1 2564.485,E2 2564.485} C_VEL
LIN {X 0,Y 166.314,Z 741.746,A -85,B 0,C 180,E1 2558.045,E2 2558.045} C_VEL
LIN {X 0,Y 180.193,Z 731.157,A -85,B 0,C 180,E1 2552.499,E2 2552.499} C_VEL
LIN {X 0,Y 193.971,Z 719.809,A -85,B 0,C 180,E1 2548.185,E2 2548.185} C_VEL
LIN {X 0,Y 208.663,Z 706.282,A -85,B 0,C 180,E1 2544.439,E2 2544.439} C_VEL
LIN {X 0,Y 223.3,Z 691.336,A -85,B 0,C 180,E1 2541.358,E2 2541.358} C_VEL
LIN {X 0,Y 237.218,Z 675.453,A -85,B 0,C 180,E1 2538.875,E2 2538.875} C_VEL
LIN {X 0,Y 250.21,Z 658.487,A -85,B 0,C 180,E1 2536.857,E2 2536.857} C_VEL
LIN {X 0,Y 263.045,Z 639.44,A -85,B 0,C 180,E1 2535.105,E2 2535.105} C_VEL
LIN {X 0,Y 273.841,Z 620.993,A -85,B 0,C 180,E1 2533.784,E2 2533.784} C_VEL
LIN {X 0,Y 283.397,Z 601.808,A -85,B 0,C 180,E1 2532.71,E2 2532.71} C_VEL
LIN {X 0,Y 292.128,Z 581.233,A -85,B 0,C 180,E1 2531.803,E2 2531.803} C_VEL
LIN {X 0,Y 299.303,Z 560.292,A -85,B 0,C 180,E1 2531.104,E2 2531.104} C_VEL
LIN {X 0,Y 305.538,Z 537.014,A -85,B 0,C 180,E1 2530.536,E2 2530.536} C_VEL
LIN {X 0,Y 309.916,Z 514.376,A -85,B 0,C 180,E1 2530.109,E2 2530.109} C_VEL
LIN {X 0,Y 321.768,Z 410.775,A -85,B 0,C 180,E1 2528.432,E2 2528.432} C_VEL
LIN {X 0,Y 324.126,Z 389.748,A -85,B 0,C 180,E1 2528.06,E2 2528.06} C_VEL
LIN {X 0,Y 323.343,Z 387.018,A -85,B 0,C 180,E1 2525.501,E2 2525.501} C_VEL
LIN {X 0,Y 323.126,Z 385.037,A -85,B 0,C 180,E1 2521.419,E2 2521.419} C_VEL
LIN {X 0,Y 324.362,Z 387.71,A -85,B 0,C 180,E1 2516.643,E2 2516.643} C_VEL
LIN {X 0,Y 324.566,Z 388.655,A -85,B 0,C 180,E1 2516.094,E2 2516.094} C_VEL
LIN {X 0,Y 316.804,Z 456.852,A -85,B 0,C 180,E1 2514.966,E2 2514.966} C_VEL
LIN {X 0,Y 315.805,Z 464.548,A -85,B 0,C 180,E1 2515.02,E2 2515.02} C_VEL
LIN {X 0,Y 312.715,Z 485.116,A -85,B 0,C 180,E1 2515.809,E2 2515.809} C_VEL
LIN {X 0,Y 311.875,Z 491.72,A -85,B 0,C 180,E1 2515.841,E2 2515.841} C_VEL
LIN {X 0,Y 307.928,Z 520.255,A -85,B 0,C 180,E1 2515.355,E2 2515.355} C_VEL
LIN {X 0,Y 303.078,Z 543.002,A -85,B 0,C 180,E1 2514.904,E2 2514.904} C_VEL
LIN {X 0,Y 296.935,Z 563.988,A -85,B 0,C 180,E1 2514.365,E2 2514.365} C_VEL
LIN {X 0,Y 288.754,Z 586.395,A -85,B 0,C 180,E1 2513.594,E2 2513.594} C_VEL
LIN {X 0,Y 279.828,Z 606.521,A -85,B 0,C 180,E1 2512.697,E2 2512.697} C_VEL
LIN {X 0,Y 269.368,Z 626.345,A -85,B 0,C 180,E1 2511.563,E2 2511.563} C_VEL
LIN {X 0,Y 257.725,Z 645.506,A -85,B 0,C 180,E1 2510.172,E2 2510.172} C_VEL
LIN {X 0,Y 245.36,Z 663.097,A -85,B 0,C 180,E1 2508.529,E2 2508.529} C_VEL
LIN {X 0,Y 231.139,Z 680.984,A -85,B 0,C 180,E1 2506.377,E2 2506.377} C_VEL
LIN {X 0,Y 216.985,Z 696.833,A -85,B 0,C 180,E1 2503.89,E2 2503.89} C_VEL
LIN {X 0,Y 202.188,Z 711.551,A -85,B 0,C 180,E1 2500.822,E2 2500.822} C_VEL
LIN {X 0,Y 186.881,Z 725.408,A -85,B 0,C 180,E1 2496.958,E2 2496.958} C_VEL
LIN {X 0,Y 172.169,Z 737.52,A -85,B 0,C 180,E1 2492.317,E2 2492.317} C_VEL
LIN {X 0,Y 158.086,Z 748.239,A -85,B 0,C 180,E1 2486.6,E2 2486.6} C_VEL
LIN {X 0,Y 145.475,Z 757.454,A -85,B 0,C 180,E1 2479.719,E2 2479.719} C_VEL
LIN {X 0,Y 134.674,Z 765.097,A -85,B 0,C 180,E1 2471.356,E2 2471.356} C_VEL
LIN {X 0,Y 126.389,Z 771.322,A -85,B 0,C 180,E1 2461.31,E2 2461.31} C_VEL
LIN {X 0,Y 121.998,Z 775.288,A -85,B 0,C 180,E1 2451.641,E2 2451.641} C_VEL
LIN {X 0,Y 120.189,Z 777.765,A -85,B 0,C 180,E1 2441.517,E2 2441.517} C_VEL
LIN {X 0,Y 120.041,Z 778.625,A -85,B 0,C 180,E1 2434.299,E2 2434.299} C_VEL
LIN {X 0,Y 120.071,Z 778.747,A -85,B 0,C 180,E1 2428.091,E2 2428.091} C_VEL
LIN {X 0,Y 120.075,Z 778.127,A -85,B 0,C 180,E1 2420.897,E2 2420.897} C_VEL
LIN {X 0,Y 120.928,Z 776.488,A -85,B 0,C 180,E1 2412.684,E2 2412.684} C_VEL
LIN {X 0,Y 124.209,Z 773.19,A -85,B 0,C 180,E1 2402.689,E2 2402.689} C_VEL
LIN {X 0,Y 130.335,Z 768.224,A -85,B 0,C 180,E1 2393.248,E2 2393.248} C_VEL
LIN {X 0,Y 139.732,Z 761.441,A -85,B 0,C 180,E1 2384.313,E2 2384.313} C_VEL
LIN {X 0,Y 151.218,Z 753.197,A -85,B 0,C 180,E1 2376.867,E2 2376.867} C_VEL
LIN {X 0,Y 164.759,Z 743.142,A -85,B 0,C 180,E1 2370.49,E2 2370.49} C_VEL
LIN {X 0,Y 179.194,Z 731.798,A -85,B 0,C 180,E1 2365.326,E2 2365.326} C_VEL
LIN {X 0,Y 194.02,Z 718.957,A -85,B 0,C 180,E1 2361.135,E2 2361.135} C_VEL
LIN {X 0,Y 210.192,Z 703.57,A -85,B 0,C 180,E1 2357.438,E2 2357.438} C_VEL
LIN {X 0,Y 225.238,Z 687.658,A -85,B 0,C 180,E1 2354.602,E2 2354.602} C_VEL
LIN {X 0,Y 239.466,Z 670.533,A -85,B 0,C 180,E1 2352.31,E2 2352.31} C_VEL
LIN {X 0,Y 253.116,Z 651.967,A -85,B 0,C 180,E1 2350.401,E2 2350.401} C_VEL
LIN {X 0,Y 265.377,Z 632.971,A -85,B 0,C 180,E1 2348.886,E2 2348.886} C_VEL
LIN {X 0,Y 276.412,Z 612.88,A -85,B 0,C 180,E1 2347.647,E2 2347.647} C_VEL
LIN {X 0,Y 286.524,Z 591.229,A -85,B 0,C 180,E1 2346.612,E2 2346.612} C_VEL
LIN {X 0,Y 294.644,Z 570.323,A -85,B 0,C 180,E1 2345.843,E2 2345.843} C_VEL
LIN {X 0,Y 301.24,Z 548.873,A -85,B 0,C 180,E1 2345.242,E2 2345.242} C_VEL
LIN {X 0,Y 306.6,Z 526.284,A -85,B 0,C 180,E1 2344.762,E2 2344.762} C_VEL
LIN {X 0,Y 310.206,Z 503.845,A -85,B 0,C 180,E1 2344.364,E2 2344.364} C_VEL
LIN {X 0,Y 322.81,Z 394.933,A -85,B 0,C 180,E1 2342.574,E2 2342.574} C_VEL
LIN {X 0,Y 321.922,Z 392.618,A -85,B 0,C 180,E1 2338.398,E2 2338.398} C_VEL
LIN {X 0,Y 322.278,Z 395.407,A -85,B 0,C 180,E1 2333.766,E2 2333.766} C_VEL
LIN {X 0,Y 322.433,Z 396.295,A -85,B 0,C 180,E1 2333.123,E2 2333.123} C_VEL
LIN {X 0,Y 308.738,Z 513.907,A -85,B 0,C 180,E1 2331.277,E2 2331.277} C_VEL
LIN {X 0,Y 304.335,Z 536.558,A -85,B 0,C 180,E1 2330.87,E2 2330.87} C_VEL
LIN {X 0,Y 298.598,Z 558.17,A -85,B 0,C 180,E1 2330.381,E2 2330.381} C_VEL
LIN {X 0,Y 291.604,Z 578.624,A -85,B 0,C 180,E1 2329.751,E2 2329.751} C_VEL
LIN {X 0,Y 282.744,Z 599.775,A -85,B 0,C 180,E1 2328.898,E2 2328.898} C_VEL
LIN {X 0,Y 273.037,Z 619.306,A -85,B 0,C 180,E1 2327.884,E2 2327.884} C_VEL
LIN {X 0,Y 262.048,Z 637.963,A -85,B 0,C 180,E1 2326.641,E2 2326.641} C_VEL
LIN {X 0,Y 249.865,Z 656.084,A -85,B 0,C 180,E1 2325.096,E2 2325.096} C_VEL
LIN {X 0,Y 237.785,Z 671.777,A -85,B 0,C 180,E1 2323.385,E2 2323.385} C_VEL
LIN {X 0,Y 223.122,Z 688.642,A -85,B 0,C 180,E1 2320.999,E2 2320.999} C_VEL
LIN {X 0,Y 208.815,Z 703.301,A -85,B 0,C 180,E1 2318.263,E2 2318.263} C_VEL
LIN {X 0,Y 194.251,Z 716.481,A -85,B 0,C 180,E1 2314.943,E2 2314.943} C_VEL
LIN {X 0,Y 178.955,Z 729.037,A -85,B 0,C 180,E1 2310.642,E2 2310.642} C_VEL
LIN {X 0,Y 165.154,Z 739.332,A -85,B 0,C 180,E1 2305.734,E2 2305.734} C_VEL
LIN {X 0,Y 152.09,Z 748.267,A -85,B 0,C 180,E1 2299.692,E2 2299.692} C_VEL
LIN {X 0,Y 140.652,Z 755.752,A -85,B 0,C 180,E1 2292.478,E2 2292.478} C_VEL
LIN {X 0,Y 131.178,Z 761.713,A -85,B 0,C 180,E1 2283.807,E2 2283.807} C_VEL
LIN {X 0,Y 124.376,Z 766.221,A -85,B 0,C 180,E1 2273.586,E2 2273.586} C_VEL
LIN {X 0,Y 121.164,Z 768.801,A -85,B 0,C 180,E1 2263.846,E2 2263.846} C_VEL
LIN {X 0,Y 120.177,Z 769.894,A -85,B 0,C 180,E1 2254.772,E2 2254.772} C_VEL
LIN {X 0,Y 120.116,Z 770.005,A -85,B 0,C 180,E1 2247.615,E2 2247.615} C_VEL
LIN {X 0,Y 120.555,Z 769.385,A -85,B 0,C 180,E1 2239.97,E2 2239.97} C_VEL
LIN {X 0,Y 122.677,Z 767.565,A -85,B 0,C 180,E1 2230.479,E2 2230.479} C_VEL
LIN {X 0,Y 127.78,Z 763.944,A -85,B 0,C 180,E1 2220.465,E2 2220.465} C_VEL
LIN {X 0,Y 136.369,Z 758.482,A -85,B 0,C 180,E1 2210.911,E2 2210.911} C_VEL
LIN {X 0,Y 146.845,Z 751.819,A -85,B 0,C 180,E1 2203.236,E2 2203.236} C_VEL
LIN {X 0,Y 159.704,Z 743.203,A -85,B 0,C 180,E1 2196.497,E2 2196.497} C_VEL
LIN {X 0,Y 173.768,Z 733.143,A -85,B 0,C 180,E1 2190.983,E2 2190.983} C_VEL
LIN {X 0,Y 187.923,Z 721.988,A -85,B 0,C 180,E1 2186.641,E2 2186.641} C_VEL
LIN {X 0,Y 203.065,Z 708.795,A -85,B 0,C 180,E1 2182.892,E2 2182.892} C_VEL
LIN {X 0,Y 217.93,Z 694.409,A -85,B 0,C 180,E1 2179.863,E2 2179.863} C_VEL
LIN {X 0,Y 232.157,Z 678.742,A -85,B 0,C 180,E1 2177.406,E2 2177.406} C_VEL
LIN {X 0,Y 246.357,Z 661.072,A -85,B 0,C 180,E1 2175.296,E2 2175.296} C_VEL
LIN {X 0,Y 258.798,Z 643.481,A -85,B 0,C 180,E1 2173.68,E2 2173.68} C_VEL
LIN {X 0,Y 270.201,Z 624.679,A -85,B 0,C 180,E1 2172.344,E2 2172.344} C_VEL
LIN {X 0,Y 280.818,Z 604.367,A -85,B 0,C 180,E1 2171.218,E2 2171.218} C_VEL
LIN {X 0,Y 289.839,Z 583.825,A -85,B 0,C 180,E1 2170.334,E2 2170.334} C_VEL
LIN {X 0,Y 297.402,Z 562.592,A -85,B 0,C 180,E1 2169.643,E2 2169.643} C_VEL
LIN {X 0,Y 303.686,Z 540.409,A -85,B 0,C 180,E1 2169.11,E2 2169.11} C_VEL
LIN {X 0,Y 308.247,Z 518.216,A -85,B 0,C 180,E1 2168.702,E2 2168.702} C_VEL
LIN {X 0,Y 312.552,Z 484.817,A -85,B 0,C 180,E1 2168.164,E2 2168.164} C_VEL
LIN {X 0,Y 322.671,Z 396.365,A -85,B 0,C 180,E1 2166.763,E2 2166.763} C_VEL
LIN {X 0,Y 322.286,Z 394.79,A -85,B 0,C 180,E1 2165.162,E2 2165.162} C_VEL
LIN {X 0,Y 322.151,Z 392.98,A -85,B 0,C 180,E1 2161.423,E2 2161.423} C_VEL
LIN {X 0,Y 323.028,Z 395.264,A -85,B 0,C 180,E1 2157.4,E2 2157.4} C_VEL
LIN {X 0,Y 311.875,Z 491.72,A -85,B 0,C 180,E1 2155.841,E2 2155.841} C_VEL
LIN {X 0,Y 310.891,Z 499.412,A -85,B 0,C 180,E1 2155.911,E2 2155.911} C_VEL
LIN {X 0,Y 307.457,Z 518.795,A -85,B 0,C 180,E1 2156.7,E2 2156.7} C_VEL
LIN {X 0,Y 305.949,Z 526.418,A -85,B 0,C 180,E1 2156.734,E2 2156.734} C_VEL
LIN {X 0,Y 300.523,Z 548.985,A -85,B 0,C 180,E1 2156.28,E2 2156.28} C_VEL
LIN {X 0,Y 294.015,Z 569.947,A -85,B 0,C 180,E1 2155.732,E2 2155.732} C_VEL
LIN {X 0,Y 285.722,Z 591.042,A -85,B 0,C 180,E1 2155.004,E2 2155.004} C_VEL
LIN {X 0,Y 275.447,Z 612.75,A -85,B 0,C 180,E1 2154.03,E2 2154.03} C_VEL
LIN {X 0,Y 264.489,Z 632.434,A -85,B 0,C 180,E1 2152.89,E2 2152.89} C_VEL
LIN {X 0,Y 252.234,Z 651.163,A -85,B 0,C 180,E1 2151.491,E2 2151.491} C_VEL
LIN {X 0,Y 238.306,Z 669.83,A -85,B 0,C 180,E1 2149.692,E2 2149.692} C_VEL
LIN {X 0,Y 224.194,Z 686.472,A -85,B 0,C 180,E1 2147.598,E2 2147.598} C_VEL
LIN {X 0,Y 209.101,Z 702.167,A -85,B 0,C 180,E1 2144.989,E2 2144.989} C_VEL
LIN {X 0,Y 193.675,Z 716.618,A -85,B 0,C 180,E1 2141.784,E2 2141.784} C_VEL
LIN {X 0,Y 178.685,Z 729.206,A -85,B 0,C 180,E1 2137.982,E2 2137.982} C_VEL
LIN {X 0,Y 162.846,Z 741.329,A -85,B 0,C 180,E1 2132.906,E2 2132.906} C_VEL
LIN {X 0,Y 148.278,Z 751.702,A -85,B 0,C 180,E1 2126.733,E2 2126.733} C_VEL
LIN {X 0,Y 135.633,Z 760.094,A -85,B 0,C 180,E1 2119.4,E2 2119.4} C_VEL
LIN {X 0,Y 124.555,Z 767.43,A -85,B 0,C 180,E1 2109.954,E2 2109.954} C_VEL
LIN {X 0,Y 117.437,Z 772.486,A -85,B 0,C 180,E1 2100.153,E2 2100.153} C_VEL
LIN {X 0,Y 113.252,Z 776.087,A -85,B 0,C 180,E1 2089.066,E2 2089.066} C_VEL
LIN {X 0,Y 112.116,Z 777.77,A -85,B 0,C 180,E1 2080.274,E2 2080.274} C_VEL
LIN {X 0,Y 112.059,Z 778.411,A -85,B 0,C 180,E1 2073.069,E2 2073.069} C_VEL
LIN {X 0,Y 112.059,Z 778.407,A -85,B 0,C 180,E1 2066.931,E2 2066.931} C_VEL
LIN {X 0,Y 112.117,Z 777.758,A -85,B 0,C 180,E1 2059.726,E2 2059.726} C_VEL
LIN {X 0,Y 113.281,Z 776.036,A -85,B 0,C 180,E1 2050.806,E2 2050.806} C_VEL
LIN {X 0,Y 117.706,Z 772.231,A -85,B 0,C 180,E1 2039.359,E2 2039.359} C_VEL
LIN {X 0,Y 124.966,Z 767.117,A -85,B 0,C 180,E1 2029.604,E2 2029.604} C_VEL
LIN {X 0,Y 135.627,Z 760.028,A -85,B 0,C 180,E1 2020.597,E2 2020.597} C_VEL
LIN {X 0,Y 148.273,Z 751.626,A -85,B 0,C 180,E1 2013.264,E2 2013.264} C_VEL
LIN {X 0,Y 162.84,Z 741.234,A -85,B 0,C 180,E1 2007.09,E2 2007.09} C_VEL
LIN {X 0,Y 178.93,Z 728.873,A -85,B 0,C 180,E1 2001.94,E2 2001.94} C_VEL
LIN {X 0,Y 194.508,Z 715.758,A -85,B 0,C 180,E1 1998.019,E2 1998.019} C_VEL
LIN {X 0,Y 209.968,Z 701.121,A -85,B 0,C 180,E1 1994.839,E2 1994.839} C_VEL
LIN {X 0,Y 225.989,Z 684.19,A -85,B 0,C 180,E1 1992.107,E2 1992.107} C_VEL
LIN {X 0,Y 239.929,Z 667.592,A -85,B 0,C 180,E1 1990.08,E2 1990.08} C_VEL
LIN {X 0,Y 252.963,Z 649.794,A -85,B 0,C 180,E1 1988.409,E2 1988.409} C_VEL
LIN {X 0,Y 265.43,Z 630.418,A -85,B 0,C 180,E1 1986.994,E2 1986.994} C_VEL
LIN {X 0,Y 275.921,Z 611.429,A -85,B 0,C 180,E1 1985.911,E2 1985.911} C_VEL
LIN {X 0,Y 286.02,Z 589.803,A -85,B 0,C 180,E1 1984.955,E2 1984.955} C_VEL
LIN {X 0,Y 294.413,Z 568.094,A -85,B 0,C 180,E1 1984.218,E2 1984.218} C_VEL
